LIN {X 0,Y 544.562,Z 1211.677,A -85,B 0,C 180,E1 25546.246,E2 25546.246} C_VEL
LIN {X 0,Y 545.068,Z 1204.229,A -85,B 0,C 180,E1 25544.028,E2 25544.028} C_VEL
LIN {X 0,Y 545.864,Z 1194.826,A -85,B 0,C 180,E1 25541.746,E2 25541.746} C_VEL
LIN {X 0,Y 546.932,Z 1184.101,A -85,B 0,C 180,E1 25539.563,E2 25539.563} C_VEL
LIN {X 0,Y 548.229,Z 1171.822,A -85,B 0,C 180,E1 25537.48,E2 25537.48} C_VEL
LIN {X 0,Y 549.884,Z 1157.402,A -85,B 0,C 180,E1 25535.392,E2 25535.392} C_VEL
LIN {X 0,Y 551.64,Z 1142.682,A -85,B 0,C 180,E1 25533.563,E2 25533.563} C_VEL
LIN {X 0,Y 553.416,Z 1127.177,A -85,B 0,C 180,E1 25531.923,E2 25531.923} C_VEL
LIN {X 0,Y 555.29,Z 1110.35,A -85,B 0,C 180,E1 25530.377,E2 25530.377} C_VEL
LIN {X 0,Y 557.037,Z 1093.4,A -85,B 0,C 180,E1 25529.051,E2 25529.051} C_VEL
LIN {X 0,Y 558.861,Z 1073.803,A -85,B 0,C 180,E1 25527.747,E2 25527.747} C_VEL
LIN {X 0,Y 560.413,Z 1054.46,A -85,B 0,C 180,E1 25526.665,E2 25526.665} C_VEL
LIN {X 0,Y 561.698,Z 1033.944,A -85,B 0,C 180,E1 25525.739,E2 25525.739} C_VEL
LIN {X 0,Y 562.756,Z 1011.905,A -85,B 0,C 180,E1 25524.95,E2 25524.95} C_VEL
LIN {X 0,Y 563.403,Z 990.948,A -85,B 0,C 180,E1 25524.379,E2 25524.379} C_VEL
LIN {X 0,Y 563.645,Z 969.284,A -85,B 0,C 180,E1 25523.981,E2 25523.981} C_VEL
LIN {X 0,Y 565.376,Z 853.6,A -85,B 0,C 180,E1 25522.448,E2 25522.448} C_VEL
LIN {X 0,Y 567.818,Z 763.974,A -85,B 0,C 180,E1 25521.099,E2 25521.099} C_VEL
LIN {X 0,Y 569.634,Z 711.383,A -85,B 0,C 180,E1 25520.211,E2 25520.211} C_VEL
LIN {X 0,Y 564.325,Z 714.5,A -85,B 0,C 180,E1 25519.789,E2 25519.789} C_VEL
LIN {X 0,Y 560.672,Z 715.375,A -85,B 0,C 180,E1 25519.441,E2 25519.441} C_VEL
LIN {X 0,Y 559.123,Z 715.198,A -85,B 0,C 180,E1 25519.252,E2 25519.252} C_VEL
LIN {X 0,Y 554.906,Z 729.11,A -85,B 0,C 180,E1 25517.706,E2 25517.706} C_VEL
LIN {X 0,Y 551.52,Z 746.313,A -85,B 0,C 180,E1 25516.035,E2 25516.035} C_VEL
LIN {X 0,Y 548.829,Z 768.841,A -85,B 0,C 180,E1 25514.104,E2 25514.104} C_VEL
LIN {X 0,Y 548.008,Z 793.1,A -85,B 0,C 180,E1 25512.18,E2 25512.18} C_VEL
LIN {X 0,Y 549.552,Z 814.095,A -85,B 0,C 180,E1 25510.568,E2 25510.568} C_VEL
LIN {X 0,Y 553.126,Z 833.312,A -85,B 0,C 180,E1 25509.117,E2 25509.117} C_VEL
LIN {X 0,Y 558.641,Z 851.04,A -85,B 0,C 180,E1 25507.793,E2 25507.793} C_VEL
LIN {X 0,Y 566.486,Z 868.661,A -85,B 0,C 180,E1 25506.502,E2 25506.502} C_VEL
LIN {X 0,Y 575.748,Z 884.402,A -85,B 0,C 180,E1 25505.375,E2 25505.375} C_VEL
LIN {X 0,Y 586.391,Z 898.731,A -85,B 0,C 180,E1 25504.381,E2 25504.381} C_VEL
LIN {X 0,Y 587.254,Z 899.863,A -85,B 0,C 180,E1 25504.305,E2 25504.305} C_VEL
LIN {X 0,Y 579.576,Z 911.271,A -85,B 0,C 180,E1 25503.697,E2 25503.697} C_VEL
LIN {X 0,Y 571.301,Z 934.87,A -85,B 0,C 180,E1 25503.762,E2 25503.762} C_VEL
LIN {X 0,Y 566.013,Z 954.731,A -85,B 0,C 180,E1 25503.715,E2 25503.715} C_VEL
LIN {X 0,Y 563.46,Z 969.81,A -85,B 0,C 180,E1 25503.539,E2 25503.539} C_VEL
LIN {X 0,Y 562.158,Z 989.948,A -85,B 0,C 180,E1 25503.128,E2 25503.128} C_VEL
LIN {X 0,Y 560.251,Z 1022.157,A -85,B 0,C 180,E1 25502.29,E2 25502.29} C_VEL
LIN {X 0,Y 558.395,Z 1051.426,A -85,B 0,C 180,E1 25501.335,E2 25501.335} C_VEL
LIN {X 0,Y 556.632,Z 1080.044,A -85,B 0,C 180,E1 25500.198,E2 25500.198} C_VEL
LIN {X 0,Y 554.956,Z 1107.84,A -85,B 0,C 180,E1 25498.874,E2 25498.874} C_VEL
LIN {X 0,Y 553.378,Z 1132.67,A -85,B 0,C 180,E1 25497.478,E2 25497.478} C_VEL
LIN {X 0,Y 551.863,Z 1155.997,A -85,B 0,C 180,E1 25495.948,E2 25495.948} C_VEL
LIN {X 0,Y 550.467,Z 1176.831,A -85,B 0,C 180,E1 25494.353,E2 25494.353} C_VEL
LIN {X 0,Y 549.066,Z 1196.682,A -85,B 0,C 180,E1 25492.588,E2 25492.588} C_VEL
LIN {X 0,Y 547.917,Z 1213.443,A -85,B 0,C 180,E1 25490.847,E2 25490.847} C_VEL
LIN {X 0,Y 546.809,Z 1229.626,A -85,B 0,C 180,E1 25488.886,E2 25488.886} C_VEL
LIN {X 0,Y 545.96,Z 1242.613,A -85,B 0,C 180,E1 25487.041,E2 25487.041} C_VEL
LIN {X 0,Y 545.256,Z 1254.791,A -85,B 0,C 180,E1 25484.986,E2 25484.986} C_VEL
LIN {X 0,Y 544.689,Z 1265.458,A -85,B 0,C 180,E1 25482.835,E2 25482.835} C_VEL
LIN {X 0,Y 544.341,Z 1274.037,A -85,B 0,C 180,E1 25480.693,E2 25480.693} C_VEL
LIN {X 0,Y 544.118,Z 1281.473,A -85,B 0,C 180,E1 25478.349,E2 25478.349} C_VEL
LIN {X 0,Y 544.015,Z 1286.703,A -85,B 0,C 180,E1 25476.092,E2 25476.092} C_VEL
LIN {X 0,Y 543.973,Z 1290.229,A -85,B 0,C 180,E1 25473.901,E2 25473.901} C_VEL
LIN {X 0,Y 543.96,Z 1292.291,A -85,B 0,C 180,E1 25471.581,E2 25471.581} C_VEL
LIN {X 0,Y 543.956,Z 1292.686,A -85,B 0,C 180,E1 25469.264,E2 25469.264} C_VEL
LIN {X 0,Y 543.956,Z 1291.533,A -85,B 0,C 180,E1 25467.051,E2 25467.051} C_VEL
LIN {X 0,Y 543.973,Z 1288.582,A -85,B 0,C 180,E1 25464.622,E2 25464.622} C_VEL
LIN {X 0,Y 544.03,Z 1284.043,A -85,B 0,C 180,E1 25462.291,E2 25462.291} C_VEL
LIN {X 0,Y 544.211,Z 1277.901,A -85,B 0,C 180,E1 25460,E2 25460} C_VEL
LIN {X 0,Y 544.557,Z 1270.094,A -85,B 0,C 180,E1 25457.704,E2 25457.704} C_VEL
LIN {X 0,Y 545.171,Z 1259.584,A -85,B 0,C 180,E1 25455.232,E2 25455.232} C_VEL
LIN {X 0,Y 546.016,Z 1247.891,A -85,B 0,C 180,E1 25452.964,E2 25452.964} C_VEL
LIN {X 0,Y 547.133,Z 1234.759,A -85,B 0,C 180,E1 25450.797,E2 25450.797} C_VEL
LIN {X 0,Y 548.623,Z 1219.348,A -85,B 0,C 180,E1 25448.624,E2 25448.624} C_VEL
LIN {X 0,Y 550.417,Z 1202.151,A -85,B 0,C 180,E1 25446.547,E2 25446.547} C_VEL
LIN {X 0,Y 552.431,Z 1184.117,A -85,B 0,C 180,E1 25444.664,E2 25444.664} C_VEL
LIN {X 0,Y 554.712,Z 1164.306,A -85,B 0,C 180,E1 25442.87,E2 25442.87} C_VEL
LIN {X 0,Y 556.979,Z 1144.891,A -85,B 0,C 180,E1 25441.361,E2 25441.361} C_VEL
LIN {X 0,Y 559.484,Z 1123.679,A -85,B 0,C 180,E1 25439.916,E2 25439.916} C_VEL
LIN {X 0,Y 562.031,Z 1101.534,A -85,B 0,C 180,E1 25438.645,E2 25438.645} C_VEL
LIN {X 0,Y 564.568,Z 1079.231,A -85,B 0,C 180,E1 25437.547,E2 25437.547} C_VEL
LIN {X 0,Y 567.05,Z 1055.53,A -85,B 0,C 180,E1 25436.599,E2 25436.599} C_VEL
LIN {X 0,Y 569.474,Z 1031.429,A -85,B 0,C 180,E1 25435.818,E2 25435.818} C_VEL
LIN {X 0,Y 571.497,Z 1007.453,A -85,B 0,C 180,E1 25435.234,E2 25435.234} C_VEL
LIN {X 0,Y 573.01,Z 980.269,A -85,B 0,C 180,E1 25434.735,E2 25434.735} C_VEL
LIN {X 0,Y 574.653,Z 963.231,A -85,B 0,C 180,E1 25434.528,E2 25434.528} C_VEL
LIN {X 0,Y 576.296,Z 952.9,A -85,B 0,C 180,E1 25434.434,E2 25434.434} C_VEL
LIN {X 0,Y 584.411,Z 939.055,A -85,B 0,C 180,E1 25433.704,E2 25433.704} C_VEL
LIN {X 0,Y 595.54,Z 921.987,A -85,B 0,C 180,E1 25432.893,E2 25432.893} C_VEL
LIN {X 0,Y 595.784,Z 921.452,A -85,B 0,C 180,E1 25432.862,E2 25432.862} C_VEL
LIN {X 0,Y 586.983,Z 910.439,A -85,B 0,C 180,E1 25431.433,E2 25431.433} C_VEL
LIN {X 0,Y 579.494,Z 897.396,A -85,B 0,C 180,E1 25429.852,E2 25429.852} C_VEL
LIN {X 0,Y 573.88,Z 882.911,A -85,B 0,C 180,E1 25428.221,E2 25428.221} C_VEL
LIN {X 0,Y 570.376,Z 867.493,A -85,B 0,C 180,E1 25426.595,E2 25426.595} C_VEL
LIN {X 0,Y 568.831,Z 850.15,A -85,B 0,C 180,E1 25424.898,E2 25424.898} C_VEL
LIN {X 0,Y 569.395,Z 830.215,A -85,B 0,C 180,E1 25423.073,E2 25423.073} C_VEL
LIN {X 0,Y 573.141,Z 791.098,A -85,B 0,C 180,E1 25419.636,E2 25419.636} C_VEL
LIN {X 0,Y 576.634,Z 756.144,A -85,B 0,C 180,E1 25416.496,E2 25416.496} C_VEL
LIN {X 0,Y 579.993,Z 723.11,A -85,B 0,C 180,E1 25413.45,E2 25413.45} C_VEL
LIN {X 0,Y 581.981,Z 702.852,A -85,B 0,C 180,E1 25411.527,E2 25411.527} C_VEL
LIN {X 0,Y 573.862,Z 683.052,A -85,B 0,C 180,E1 25408.517,E2 25408.517} C_VEL
LIN {X 0,Y 566.014,Z 664.757,A -85,B 0,C 180,E1 25405.534,E2 25405.534} C_VEL
LIN {X 0,Y 558.284,Z 647.753,A -85,B 0,C 180,E1 25402.537,E2 25402.537} C_VEL
LIN {X 0,Y 552.535,Z 635.448,A -85,B 0,C 180,E1 25400.221,E2 25400.221} C_VEL
LIN {X 0,Y 549.142,Z 628.134,A -85,B 0,C 180,E1 25398.801,E2 25398.801} C_VEL
LIN {X 0,Y 547.28,Z 624.068,A -85,B 0,C 180,E1 25397.985,E2 25397.985} C_VEL
LIN {X 0,Y 545.723,Z 620.923,A -85,B 0,C 180,E1 25397.34,E2 25397.34} C_VEL
LIN {X 0,Y 545.56,Z 620.018,A -85,B 0,C 180,E1 25397.162,E2 25397.162} C_VEL
LIN {X 0,Y 545.561,Z 620.023,A -85,B 0,C 180,E1 25393.676,E2 25393.676} C_VEL
LIN {X 0,Y 545.551,Z 620.018,A -85,B 0,C 180,E1 25390.347,E2 25390.347} C_VEL
LIN {X 0,Y 545.565,Z 620.021,A -85,B 0,C 180,E1 25386.948,E2 25386.948} C_VEL
LIN {X 0,Y 545.556,Z 620.018,A -85,B 0,C 180,E1 25383.573,E2 25383.573} C_VEL
LIN {X 0,Y 545.556,Z 620.024,A -85,B 0,C 180,E1 25380.21,E2 25380.21} C_VEL
LIN {X 0,Y 545.55,Z 620.025,A -85,B 0,C 180,E1 25376.848,E2 25376.848} C_VEL
LIN {X 0,Y 545.559,Z 620.021,A -85,B 0,C 180,E1 25373.475,E2 25373.475} C_VEL
LIN {X 0,Y 545.558,Z 620.018,A -85,B 0,C 180,E1 25369.973,E2 25369.973} C_VEL
LIN {X 0,Y 545.56,Z 620.016,A -85,B 0,C 180,E1 25366.54,E2 25366.54} C_VEL
LIN {X 0,Y 545.551,Z 620.018,A -85,B 0,C 180,E1 25363.277,E2 25363.277} C_VEL
LIN {X 0,Y 545.563,Z 620.017,A -85,B 0,C 180,E1 25359.957,E2 25359.957} C_VEL
LIN {X 0,Y 545.562,Z 620.016,A -85,B 0,C 180,E1 25356.565,E2 25356.565} C_VEL
LIN {X 0,Y 545.555,Z 620.015,A -85,B 0,C 180,E1 25353.193,E2 25353.193} C_VEL
LIN {X 0,Y 545.551,Z 620.019,A -85,B 0,C 180,E1 25349.855,E2 25349.855} C_VEL
LIN {X 0,Y 545.558,Z 620.022,A -85,B 0,C 180,E1 25346.499,E2 25346.499} C_VEL
LIN {X 0,Y 545.561,Z 620.023,A -85,B 0,C 180,E1 25343.04,E2 25343.04} C_VEL
LIN {X 0,Y 545.564,Z 620.024,A -85,B 0,C 180,E1 25339.676,E2 25339.676} C_VEL
LIN {X 0,Y 545.549,Z 619.992,A -85,B 0,C 180,E1 25336.293,E2 25336.293} C_VEL
LIN {X 0,Y 545.561,Z 620.016,A -85,B 0,C 180,E1 25332.981,E2 25332.981} C_VEL
LIN {X 0,Y 545.567,Z 620.029,A -85,B 0,C 180,E1 25329.625,E2 25329.625} C_VEL
LIN {X 0,Y 545.579,Z 620.17,A -85,B 0,C 180,E1 25326.359,E2 25326.359} C_VEL
LIN {X 0,Y 554.088,Z 644.386,A -85,B 0,C 180,E1 25324.075,E2 25324.075} C_VEL
LIN {X 0,Y 559.543,Z 662.583,A -85,B 0,C 180,E1 25322.416,E2 25322.416} C_VEL
LIN {X 0,Y 558.089,Z 702.519,A -85,B 0,C 180,E1 25319.516,E2 25319.516} C_VEL
LIN {X 0,Y 556.154,Z 749.591,A -85,B 0,C 180,E1 25316.075,E2 25316.075} C_VEL
LIN {X 0,Y 554.34,Z 796.346,A -85,B 0,C 180,E1 25312.704,E2 25312.704} C_VEL
LIN {X 0,Y 553.05,Z 840.958,A -85,B 0,C 180,E1 25309.618,E2 25309.618} C_VEL
LIN {X 0,Y 553.037,Z 845.924,A -85,B 0,C 180,E1 25309.313,E2 25309.313} C_VEL
LIN {X 0,Y 553.774,Z 853.842,A -85,B 0,C 180,E1 25309.176,E2 25309.176} C_VEL
LIN {X 0,Y 553.745,Z 856.037,A -85,B 0,C 180,E1 25309.148,E2 25309.148} C_VEL
LIN {X 0,Y 552.713,Z 863.711,A -85,B 0,C 180,E1 25309.083,E2 25309.083} C_VEL
LIN {X 0,Y 546.531,Z 884.049,A -85,B 0,C 180,E1 25309.045,E2 25309.045} C_VEL
LIN {X 0,Y 545.779,Z 890.637,A -85,B 0,C 180,E1 25308.984,E2 25308.984} C_VEL
LIN {X 0,Y 544.332,Z 1016.575,A -85,B 0,C 180,E1 25307.282,E2 25307.282} C_VEL
LIN {X 0,Y 544.07,Z 1034.06,A -85,B 0,C 180,E1 25306.854,E2 25306.854} C_VEL
LIN {X 0,Y 543.55,Z 1050.898,A -85,B 0,C 180,E1 25306.235,E2 25306.235} C_VEL
LIN {X 0,Y 542.849,Z 1067.086,A -85,B 0,C 180,E1 25305.434,E2 25305.434} C_VEL
LIN {X 0,Y 542.02,Z 1082.23,A -85,B 0,C 180,E1 25304.474,E2 25304.474} C_VEL
LIN {X 0,Y 541.114,Z 1096.279,A -85,B 0,C 180,E1 25303.353,E2 25303.353} C_VEL
LIN {X 0,Y 540.183,Z 1109.272,A -85,B 0,C 180,E1 25302.072,E2 25302.072} C_VEL
LIN {X 0,Y 539.316,Z 1120.771,A -85,B 0,C 180,E1 25300.683,E2 25300.683} C_VEL
LIN {X 0,Y 538.552,Z 1130.856,A -85,B 0,C 180,E1 25299.186,E2 25299.186} C_VEL
LIN {X 0,Y 537.911,Z 1139.49,A -85,B 0,C 180,E1 25297.582,E2 25297.582} C_VEL
LIN {X 0,Y 537.417,Z 1146.684,A -85,B 0,C 180,E1 25295.872,E2 25295.872} C_VEL
LIN {X 0,Y 537.07,Z 1152.376,A -85,B 0,C 180,E1 25294.055,E2 25294.055} C_VEL
LIN {X 0,Y 536.865,Z 1156.258,A -85,B 0,C 180,E1 25292.24,E2 25292.24} C_VEL
LIN {X 0,Y 536.762,Z 1158.468,A -85,B 0,C 180,E1 25290.319,E2 25290.319} C_VEL
LIN {X 0,Y 536.741,Z 1158.887,A -85,B 0,C 180,E1 25288.397,E2 25288.397} C_VEL
LIN {X 0,Y 536.82,Z 1157.529,A -85,B 0,C 180,E1 25286.475,E2 25286.475} C_VEL
LIN {X 0,Y 536.987,Z 1154.493,A -85,B 0,C 180,E1 25284.657,E2 25284.657} C_VEL
LIN {X 0,Y 537.286,Z 1149.689,A -85,B 0,C 180,E1 25282.836,E2 25282.836} C_VEL
LIN {X 0,Y 537.745,Z 1142.99,A -85,B 0,C 180,E1 25281.013,E2 25281.013} C_VEL
LIN {X 0,Y 538.329,Z 1135.257,A -85,B 0,C 180,E1 25279.403,E2 25279.403} C_VEL
LIN {X 0,Y 539.094,Z 1125.43,A -85,B 0,C 180,E1 25277.792,E2 25277.792} C_VEL
LIN {X 0,Y 539.999,Z 1114.033,A -85,B 0,C 180,E1 25276.289,E2 25276.289} C_VEL
LIN {X 0,Y 540.962,Z 1101.428,A -85,B 0,C 180,E1 25274.939,E2 25274.939} C_VEL
LIN {X 0,Y 541.899,Z 1087.841,A -85,B 0,C 180,E1 25273.766,E2 25273.766} C_VEL
LIN {X 0,Y 542.778,Z 1073.195,A -85,B 0,C 180,E1 25272.746,E2 25272.746} C_VEL
LIN {X 0,Y 543.555,Z 1057.58,A -85,B 0,C 180,E1 25271.886,E2 25271.886} C_VEL
LIN {X 0,Y 544.156,Z 1041.565,A -85,B 0,C 180,E1 25271.213,E2 25271.213} C_VEL
LIN {X 0,Y 544.545,Z 1024.25,A -85,B 0,C 180,E1 25270.701,E2 25270.701} C_VEL
LIN {X 0,Y 544.693,Z 1004.749,A -85,B 0,C 180,E1 25270.351,E2 25270.351} C_VEL
LIN {X 0,Y 546.455,Z 851.134,A -85,B 0,C 180,E1 25268.298,E2 25268.298} C_VEL
LIN {X 0,Y 545.809,Z 845.842,A -85,B 0,C 180,E1 25268.167,E2 25268.167} C_VEL
LIN {X 0,Y 547.153,Z 801.476,A -85,B 0,C 180,E1 25265.087,E2 25265.087} C_VEL
LIN {X 0,Y 548.938,Z 757.8,A -85,B 0,C 180,E1 25261.909,E2 25261.909} C_VEL
LIN {X 0,Y 550.971,Z 712.063,A -85,B 0,C 180,E1 25258.534,E2 25258.534} C_VEL
LIN {X 0,Y 552.718,Z 669.961,A -85,B 0,C 180,E1 25255.442,E2 25255.442} C_VEL
LIN {X 0,Y 552.763,Z 665.3,A -85,B 0,C 180,E1 25255.094,E2 25255.094} C_VEL
LIN {X 0,Y 545.767,Z 643.324,A -85,B 0,C 180,E1 25253.015,E2 25253.015} C_VEL
LIN {X 0,Y 538.244,Z 623.221,A -85,B 0,C 180,E1 25251.028,E2 25251.028} C_VEL
LIN {X 0,Y 537.625,Z 620.99,A -85,B 0,C 180,E1 25250.81,E2 25250.81} C_VEL
LIN {X 0,Y 537.624,Z 621.01,A -85,B 0,C 180,E1 25247.391,E2 25247.391} C_VEL
LIN {X 0,Y 537.619,Z 621.012,A -85,B 0,C 180,E1 25243.926,E2 25243.926} C_VEL
LIN {X 0,Y 537.636,Z 621.101,A -85,B 0,C 180,E1 25241.577,E2 25241.577} C_VEL
LIN {X 0,Y 539.132,Z 624.777,A -85,B 0,C 180,E1 25240.988,E2 25240.988} C_VEL
LIN {X 0,Y 544.561,Z 636.539,A -85,B 0,C 180,E1 25239.145,E2 25239.145} C_VEL
LIN {X 0,Y 562.473,Z 662.364,A -85,B 0,C 180,E1 25237.043,E2 25237.043} C_VEL
LIN {X 0,Y 572.59,Z 677.716,A -85,B 0,C 180,E1 25235.923,E2 25235.923} C_VEL
LIN {X 0,Y 563.214,Z 919.475,A -85,B 0,C 180,E1 25232.101,E2 25232.101} C_VEL
LIN {X 0,Y 561.649,Z 966.293,A -85,B 0,C 180,E1 25231.336,E2 25231.336} C_VEL
LIN {X 0,Y 560.501,Z 989.145,A -85,B 0,C 180,E1 25230.77,E2 25230.77} C_VEL
LIN {X 0,Y 559.003,Z 1011.643,A -85,B 0,C 180,E1 25230.032,E2 25230.032} C_VEL
LIN {X 0,Y 557.268,Z 1033.005,A -85,B 0,C 180,E1 25229.153,E2 25229.153} C_VEL
LIN {X 0,Y 555.198,Z 1053.829,A -85,B 0,C 180,E1 25228.096,E2 25228.096} C_VEL
LIN {X 0,Y 552.898,Z 1075.118,A -85,B 0,C 180,E1 25226.804,E2 25226.804} C_VEL
LIN {X 0,Y 550.629,Z 1094.218,A -85,B 0,C 180,E1 25225.434,E2 25225.434} C_VEL
LIN {X 0,Y 548.259,Z 1112.608,A -85,B 0,C 180,E1 25223.883,E2 25223.883} C_VEL
LIN {X 0,Y 545.977,Z 1130.204,A -85,B 0,C 180,E1 25222.164,E2 25222.164} C_VEL
LIN {X 0,Y 543.939,Z 1145.349,A -85,B 0,C 180,E1 25220.443,E2 25220.443} C_VEL
LIN {X 0,Y 541.915,Z 1160.932,A -85,B 0,C 180,E1 25218.392,E2 25218.392} C_VEL
LIN {X 0,Y 540.25,Z 1174.381,A -85,B 0,C 180,E1 25216.339,E2 25216.339} C_VEL
LIN {X 0,Y 538.865,Z 1186.313,A -85,B 0,C 180,E1 25214.178,E2 25214.178} C_VEL
LIN {X 0,Y 537.78,Z 1196.995,A -85,B 0,C 180,E1 25211.91,E2 25211.91} C_VEL
LIN {X 0,Y 537.051,Z 1205.44,A -85,B 0,C 180,E1 25209.754,E2 25209.754} C_VEL
LIN {X 0,Y 536.512,Z 1213.345,A -85,B 0,C 180,E1 25207.281,E2 25207.281} C_VEL
LIN {X 0,Y 536.226,Z 1218.992,A -85,B 0,C 180,E1 25205.028,E2 25205.028} C_VEL
LIN {X 0,Y 536.064,Z 1223.49,A -85,B 0,C 180,E1 25202.566,E2 25202.566} C_VEL
LIN {X 0,Y 536.028,Z 1226.336,A -85,B 0,C 180,E1 25200.214,E2 25200.214} C_VEL
LIN {X 0,Y 535.991,Z 1227.612,A -85,B 0,C 180,E1 25197.862,E2 25197.862} C_VEL
LIN {X 0,Y 535.993,Z 1227.555,A -85,B 0,C 180,E1 25195.506,E2 25195.506} C_VEL
LIN {X 0,Y 536.023,Z 1225.893,A -85,B 0,C 180,E1 25193.143,E2 25193.143} C_VEL
LIN {X 0,Y 536.112,Z 1222.854,A -85,B 0,C 180,E1 25190.77,E2 25190.77} C_VEL
LIN {X 0,Y 536.279,Z 1218.382,A -85,B 0,C 180,E1 25188.492,E2 25188.492} C_VEL
LIN {X 0,Y 536.653,Z 1211.807,A -85,B 0,C 180,E1 25185.983,E2 25185.983} C_VEL
LIN {X 0,Y 537.235,Z 1204.125,A -85,B 0,C 180,E1 25183.678,E2 25183.678} C_VEL
LIN {X 0,Y 538.089,Z 1194.661,A -85,B 0,C 180,E1 25181.389,E2 25181.389} C_VEL
LIN {X 0,Y 539.201,Z 1184.229,A -85,B 0,C 180,E1 25179.256,E2 25179.256} C_VEL
LIN {X 0,Y 540.599,Z 1171.911,A -85,B 0,C 180,E1 25177.144,E2 25177.144} C_VEL
LIN {X 0,Y 542.265,Z 1158.093,A -85,B 0,C 180,E1 25175.124,E2 25175.124} C_VEL
LIN {X 0,Y 544.124,Z 1143.344,A -85,B 0,C 180,E1 25173.264,E2 25173.264} C_VEL
LIN {X 0,Y 546.025,Z 1127.486,A -85,B 0,C 180,E1 25171.568,E2 25171.568} C_VEL
LIN {X 0,Y 548.147,Z 1109.199,A -85,B 0,C 180,E1 25169.892,E2 25169.892} C_VEL
LIN {X 0,Y 550.104,Z 1091.165,A -85,B 0,C 180,E1 25168.483,E2 25168.483} C_VEL
LIN {X 0,Y 551.853,Z 1072.399,A -85,B 0,C 180,E1 25167.259,E2 25167.259} C_VEL
LIN {X 0,Y 553.498,Z 1051.713,A -85,B 0,C 180,E1 25166.13,E2 25166.13} C_VEL
LIN {X 0,Y 554.841,Z 1031.303,A -85,B 0,C 180,E1 25165.224,E2 25165.224} C_VEL
LIN {X 0,Y 555.771,Z 1010.369,A -85,B 0,C 180,E1 25164.503,E2 25164.503} C_VEL
LIN {X 0,Y 556.37,Z 988.036,A -85,B 0,C 180,E1 25163.928,E2 25163.928} C_VEL
LIN {X 0,Y 556.586,Z 965.593,A -85,B 0,C 180,E1 25163.54,E2 25163.54} C_VEL
LIN {X 0,Y 558.266,Z 867.649,A -85,B 0,C 180,E1 25162.215,E2 25162.215} C_VEL
LIN {X 0,Y 560.827,Z 781.835,A -85,B 0,C 180,E1 25160.892,E2 25160.892} C_VEL
LIN {X 0,Y 563.225,Z 722.74,A -85,B 0,C 180,E1 25159.87,E2 25159.87} C_VEL
LIN {X 0,Y 559.432,Z 723.517,A -85,B 0,C 180,E1 25159.51,E2 25159.51} C_VEL
LIN {X 0,Y 553.862,Z 727.441,A -85,B 0,C 180,E1 25158.993,E2 25158.993} C_VEL
LIN {X 0,Y 550.494,Z 728.74,A -85,B 0,C 180,E1 25158.605,E2 25158.605} C_VEL
LIN {X 0,Y 549.002,Z 728.818,A -85,B 0,C 180,E1 25158.387,E2 25158.387} C_VEL
LIN {X 0,Y 545.176,Z 744.683,A -85,B 0,C 180,E1 25156.731,E2 25156.731} C_VEL
LIN {X 0,Y 542.101,Z 764.837,A -85,B 0,C 180,E1 25154.879,E2 25154.879} C_VEL
LIN {X 0,Y 540.482,Z 788.554,A -85,B 0,C 180,E1 25152.895,E2 25152.895} C_VEL
LIN {X 0,Y 541.18,Z 809.258,A -85,B 0,C 180,E1 25151.238,E2 25151.238} C_VEL
LIN {X 0,Y 543.953,Z 828.754,A -85,B 0,C 180,E1 25149.71,E2 25149.71} C_VEL
LIN {X 0,Y 548.863,Z 847.38,A -85,B 0,C 180,E1 25148.273,E2 25148.273} C_VEL
LIN {X 0,Y 555.897,Z 865.129,A -85,B 0,C 180,E1 25146.926,E2 25146.926} C_VEL
LIN {X 0,Y 564.621,Z 881.535,A -85,B 0,C 180,E1 25145.712,E2 25145.712} C_VEL
LIN {X 0,Y 574.804,Z 896.536,A -85,B 0,C 180,E1 25144.634,E2 25144.634} C_VEL
LIN {X 0,Y 577.615,Z 900.54,A -85,B 0,C 180,E1 25144.357,E2 25144.357} C_VEL
LIN {X 0,Y 574.007,Z 906.053,A -85,B 0,C 180,E1 25144.075,E2 25144.075} C_VEL
LIN {X 0,Y 564.767,Z 932.57,A -85,B 0,C 180,E1 25144.167,E2 25144.167} C_VEL
LIN {X 0,Y 559.323,Z 952.643,A -85,B 0,C 180,E1 25144.117,E2 25144.117} C_VEL
LIN {X 0,Y 556.547,Z 967.971,A -85,B 0,C 180,E1 25143.939,E2 25143.939} C_VEL
LIN {X 0,Y 555.208,Z 984.466,A -85,B 0,C 180,E1 25143.603,E2 25143.603} C_VEL
LIN {X 0,Y 553.15,Z 1017.086,A -85,B 0,C 180,E1 25142.748,E2 25142.748} C_VEL
LIN {X 0,Y 551.133,Z 1046.801,A -85,B 0,C 180,E1 25141.776,E2 25141.776} C_VEL
LIN {X 0,Y 549.282,Z 1075.281,A -85,B 0,C 180,E1 25140.645,E2 25140.645} C_VEL
LIN {X 0,Y 547.548,Z 1102.102,A -85,B 0,C 180,E1 25139.379,E2 25139.379} C_VEL
LIN {X 0,Y 545.849,Z 1128.091,A -85,B 0,C 180,E1 25137.934,E2 25137.934} C_VEL
LIN {X 0,Y 544.224,Z 1152.54,A -85,B 0,C 180,E1 25136.341,E2 25136.341} C_VEL
LIN {X 0,Y 542.747,Z 1173.837,A -85,B 0,C 180,E1 25134.722,E2 25134.722} C_VEL
LIN {X 0,Y 541.3,Z 1194,A -85,B 0,C 180,E1 25132.941,E2 25132.941} C_VEL
LIN {X 0,Y 540.13,Z 1210.759,A -85,B 0,C 180,E1 25131.219,E2 25131.219} C_VEL
LIN {X 0,Y 539.005,Z 1226.92,A -85,B 0,C 180,E1 25129.282,E2 25129.282} C_VEL
LIN {X 0,Y 538.056,Z 1241.043,A -85,B 0,C 180,E1 25127.299,E2 25127.299} C_VEL
LIN {X 0,Y 537.314,Z 1253.479,A -85,B 0,C 180,E1 25125.213,E2 25125.213} C_VEL
LIN {X 0,Y 536.73,Z 1264.436,A -85,B 0,C 180,E1 25123.013,E2 25123.013} C_VEL
LIN {X 0,Y 536.367,Z 1273.129,A -85,B 0,C 180,E1 25120.854,E2 25120.854} C_VEL
LIN {X 0,Y 536.145,Z 1280.396,A -85,B 0,C 180,E1 25118.582,E2 25118.582} C_VEL
LIN {X 0,Y 536.036,Z 1285.812,A -85,B 0,C 180,E1 25116.32,E2 25116.32} C_VEL
LIN {X 0,Y 535.988,Z 1289.677,A -85,B 0,C 180,E1 25113.959,E2 25113.959} C_VEL
LIN {X 0,Y 535.978,Z 1291.733,A -85,B 0,C 180,E1 25111.712,E2 25111.712} C_VEL
LIN {X 0,Y 535.97,Z 1292.217,A -85,B 0,C 180,E1 25109.253,E2 25109.253} C_VEL
LIN {X 0,Y 535.968,Z 1291.077,A -85,B 0,C 180,E1 25107.007,E2 25107.007} C_VEL
LIN {X 0,Y 535.979,Z 1288.087,A -85,B 0,C 180,E1 25104.542,E2 25104.542} C_VEL
LIN {X 0,Y 536.036,Z 1283.513,A -85,B 0,C 180,E1 25102.175,E2 25102.175} C_VEL
LIN {X 0,Y 536.234,Z 1277.177,A -85,B 0,C 180,E1 25099.798,E2 25099.798} C_VEL
LIN {X 0,Y 536.587,Z 1269.432,A -85,B 0,C 180,E1 25097.518,E2 25097.518} C_VEL
LIN {X 0,Y 537.237,Z 1258.85,A -85,B 0,C 180,E1 25095.006,E2 25095.006} C_VEL
LIN {X 0,Y 538.181,Z 1246.475,A -85,B 0,C 180,E1 25092.597,E2 25092.597} C_VEL
LIN {X 0,Y 539.379,Z 1233.108,A -85,B 0,C 180,E1 25090.397,E2 25090.397} C_VEL
LIN {X 0,Y 540.965,Z 1217.481,A -85,B 0,C 180,E1 25088.193,E2 25088.193} C_VEL
LIN {X 0,Y 543.005,Z 1199.051,A -85,B 0,C 180,E1 25085.971,E2 25085.971} C_VEL
LIN {X 0,Y 545.361,Z 1178.845,A -85,B 0,C 180,E1 25083.896,E2 25083.896} C_VEL
LIN {X 0,Y 547.773,Z 1158.882,A -85,B 0,C 180,E1 25082.143,E2 25082.143} C_VEL
LIN {X 0,Y 550.131,Z 1139.735,A -85,B 0,C 180,E1 25080.673,E2 25080.673} C_VEL
LIN {X 0,Y 552.94,Z 1116.823,A -85,B 0,C 180,E1 25079.161,E2 25079.161} C_VEL
LIN {X 0,Y 555.352,Z 1097.015,A -85,B 0,C 180,E1 25078.042,E2 25078.042} C_VEL
LIN {X 0,Y 558.237,Z 1071.944,A -85,B 0,C 180,E1 25076.851,E2 25076.851} C_VEL
LIN {X 0,Y 560.724,Z 1049.643,A -85,B 0,C 180,E1 25075.985,E2 25075.985} C_VEL
LIN {X 0,Y 563.233,Z 1024.721,A -85,B 0,C 180,E1 25075.219,E2 25075.219} C_VEL
LIN {X 0,Y 565.241,Z 1001.127,A -85,B 0,C 180,E1 25074.661,E2 25074.661} C_VEL
LIN {X 0,Y 566.987,Z 972.381,A -85,B 0,C 180,E1 25074.169,E2 25074.169} C_VEL
LIN {X 0,Y 569.907,Z 951.51,A -85,B 0,C 180,E1 25073.971,E2 25073.971} C_VEL
LIN {X 0,Y 578.073,Z 937.676,A -85,B 0,C 180,E1 25073.242,E2 25073.242} C_VEL
LIN {X 0,Y 586.981,Z 923.541,A -85,B 0,C 180,E1 25072.543,E2 25072.543} C_VEL
LIN {X 0,Y 578.464,Z 912.034,A -85,B 0,C 180,E1 25071.063,E2 25071.063} C_VEL
LIN {X 0,Y 571.261,Z 898.435,A -85,B 0,C 180,E1 25069.433,E2 25069.433} C_VEL
LIN {X 0,Y 566.009,Z 883.482,A -85,B 0,C 180,E1 25067.748,E2 25067.748} C_VEL
LIN {X 0,Y 562.857,Z 867.576,A -85,B 0,C 180,E1 25066.084,E2 25066.084} C_VEL
LIN {X 0,Y 561.725,Z 849.486,A -85,B 0,C 180,E1 25064.313,E2 25064.313} C_VEL
LIN {X 0,Y 562.737,Z 828.652,A -85,B 0,C 180,E1 25062.418,E2 25062.418} C_VEL
LIN {X 0,Y 566.478,Z 791.738,A -85,B 0,C 180,E1 25059.137,E2 25059.137} C_VEL
LIN {X 0,Y 570.12,Z 756.97,A -85,B 0,C 180,E1 25055.982,E2 25055.982} C_VEL
LIN {X 0,Y 573.674,Z 723.339,A -85,B 0,C 180,E1 25052.853,E2 25052.853} C_VEL
LIN {X 0,Y 575.329,Z 706.673,A -85,B 0,C 180,E1 25051.25,E2 25051.25} C_VEL
LIN {X 0,Y 567.44,Z 687.409,A -85,B 0,C 180,E1 25048.295,E2 25048.295} C_VEL
LIN {X 0,Y 559.754,Z 669.424,A -85,B 0,C 180,E1 25045.334,E2 25045.334} C_VEL
LIN {X 0,Y 552.186,Z 652.634,A -85,B 0,C 180,E1 25042.35,E2 25042.35} C_VEL
LIN {X 0,Y 545.541,Z 638.08,A -85,B 0,C 180,E1 25039.598,E2 25039.598} C_VEL
LIN {X 0,Y 541.117,Z 628.994,A -85,B 0,C 180,E1 25037.752,E2 25037.752} C_VEL
LIN {X 0,Y 539.24,Z 624.931,A -85,B 0,C 180,E1 25036.925,E2 25036.925} C_VEL
LIN {X 0,Y 537.684,Z 621.394,A -85,B 0,C 180,E1 25036.197,E2 25036.197} C_VEL
LIN {X 0,Y 537.625,Z 621.014,A -85,B 0,C 180,E1 25036.088,E2 25036.088} C_VEL
LIN {X 0,Y 537.612,Z 621.007,A -85,B 0,C 180,E1 25032.678,E2 25032.678} C_VEL
LIN {X 0,Y 537.611,Z 621.013,A -85,B 0,C 180,E1 25029.312,E2 25029.312} C_VEL
LIN {X 0,Y 537.616,Z 621.004,A -85,B 0,C 180,E1 25025.978,E2 25025.978} C_VEL
LIN {X 0,Y 537.622,Z 621.013,A -85,B 0,C 180,E1 25022.452,E2 25022.452} C_VEL
LIN {X 0,Y 537.629,Z 621.008,A -85,B 0,C 180,E1 25019.041,E2 25019.041} C_VEL
LIN {X 0,Y 537.628,Z 621.005,A -85,B 0,C 180,E1 25015.52,E2 25015.52} C_VEL
LIN {X 0,Y 537.623,Z 621.009,A -85,B 0,C 180,E1 25012.089,E2 25012.089} C_VEL
LIN {X 0,Y 537.612,Z 621.013,A -85,B 0,C 180,E1 25008.63,E2 25008.63} C_VEL
LIN {X 0,Y 537.613,Z 621.013,A -85,B 0,C 180,E1 25005.238,E2 25005.238} C_VEL
LIN {X 0,Y 537.624,Z 621.013,A -85,B 0,C 180,E1 25001.793,E2 25001.793} C_VEL
LIN {X 0,Y 537.633,Z 621.013,A -85,B 0,C 180,E1 24998.393,E2 24998.393} C_VEL
LIN {X 0,Y 537.63,Z 621.015,A -85,B 0,C 180,E1 24994.91,E2 24994.91} C_VEL
LIN {X 0,Y 537.629,Z 621.011,A -85,B 0,C 180,E1 24991.377,E2 24991.377} C_VEL
LIN {X 0,Y 537.617,Z 621.01,A -85,B 0,C 180,E1 24987.99,E2 24987.99} C_VEL
LIN {X 0,Y 537.611,Z 621.004,A -85,B 0,C 180,E1 24984.66,E2 24984.66} C_VEL
LIN {X 0,Y 537.614,Z 621.004,A -85,B 0,C 180,E1 24981.324,E2 24981.324} C_VEL
LIN {X 0,Y 537.623,Z 620.993,A -85,B 0,C 180,E1 24977.905,E2 24977.905} C_VEL
LIN {X 0,Y 537.627,Z 621.009,A -85,B 0,C 180,E1 24974.424,E2 24974.424} C_VEL
LIN {X 0,Y 537.612,Z 620.993,A -85,B 0,C 180,E1 24970.965,E2 24970.965} C_VEL
LIN {X 0,Y 537.627,Z 620.995,A -85,B 0,C 180,E1 24967.589,E2 24967.589} C_VEL
LIN {X 0,Y 537.629,Z 621.126,A -85,B 0,C 180,E1 24966.819,E2 24966.819} C_VEL
LIN {X 0,Y 546.478,Z 646.011,A -85,B 0,C 180,E1 24964.426,E2 24964.426} C_VEL
LIN {X 0,Y 552.273,Z 665.108,A -85,B 0,C 180,E1 24962.66,E2 24962.66} C_VEL
LIN {X 0,Y 550.7,Z 706.294,A -85,B 0,C 180,E1 24959.652,E2 24959.652} C_VEL
LIN {X 0,Y 548.676,Z 752.788,A -85,B 0,C 180,E1 24956.225,E2 24956.225} C_VEL
LIN {X 0,Y 546.784,Z 800.786,A -85,B 0,C 180,E1 24952.751,E2 24952.751} C_VEL
LIN {X 0,Y 545.485,Z 846.351,A -85,B 0,C 180,E1 24949.607,E2 24949.607} C_VEL
LIN {X 0,Y 546.275,Z 854.693,A -85,B 0,C 180,E1 24949.46,E2 24949.46} C_VEL
LIN {X 0,Y 545.779,Z 890.637,A -85,B 0,C 180,E1 24948.984,E2 24948.984} C_VEL
LIN {X 0,Y 544.785,Z 898.31,A -85,B 0,C 180,E1 24948.917,E2 24948.917} C_VEL
LIN {X 0,Y 538.598,Z 918.647,A -85,B 0,C 180,E1 24948.876,E2 24948.876} C_VEL
LIN {X 0,Y 537.817,Z 925.236,A -85,B 0,C 180,E1 24948.815,E2 24948.815} C_VEL
LIN {X 0,Y 536.755,Z 1017.576,A -85,B 0,C 180,E1 24947.542,E2 24947.542} C_VEL
LIN {X 0,Y 536.485,Z 1035.069,A -85,B 0,C 180,E1 24947.107,E2 24947.107} C_VEL
LIN {X 0,Y 535.936,Z 1052.106,A -85,B 0,C 180,E1 24946.47,E2 24946.47} C_VEL
LIN {X 0,Y 535.209,Z 1068.194,A -85,B 0,C 180,E1 24945.66,E2 24945.66} C_VEL
LIN {X 0,Y 534.347,Z 1083.311,A -85,B 0,C 180,E1 24944.686,E2 24944.686} C_VEL
LIN {X 0,Y 533.401,Z 1097.328,A -85,B 0,C 180,E1 24943.55,E2 24943.55} C_VEL
LIN {X 0,Y 532.428,Z 1110.307,A -85,B 0,C 180,E1 24942.25,E2 24942.25} C_VEL
LIN {X 0,Y 531.52,Z 1121.793,A -85,B 0,C 180,E1 24940.841,E2 24940.841} C_VEL
LIN {X 0,Y 530.717,Z 1131.867,A -85,B 0,C 180,E1 24939.323,E2 24939.323} C_VEL
LIN {X 0,Y 530.041,Z 1140.486,A -85,B 0,C 180,E1 24937.696,E2 24937.696} C_VEL
LIN {X 0,Y 529.518,Z 1147.671,A -85,B 0,C 180,E1 24935.96,E2 24935.96} C_VEL
LIN {X 0,Y 529.148,Z 1153.355,A -85,B 0,C 180,E1 24934.116,E2 24934.116} C_VEL
LIN {X 0,Y 528.93,Z 1157.227,A -85,B 0,C 180,E1 24932.274,E2 24932.274} C_VEL
LIN {X 0,Y 528.82,Z 1159.427,A -85,B 0,C 180,E1 24930.324,E2 24930.324} C_VEL
LIN {X 0,Y 528.799,Z 1159.838,A -85,B 0,C 180,E1 24928.373,E2 24928.373} C_VEL
LIN {X 0,Y 528.885,Z 1158.471,A -85,B 0,C 180,E1 24926.422,E2 24926.422} C_VEL
LIN {X 0,Y 529.065,Z 1155.424,A -85,B 0,C 180,E1 24924.576,E2 24924.576} C_VEL
LIN {X 0,Y 529.387,Z 1150.611,A -85,B 0,C 180,E1 24922.728,E2 24922.728} C_VEL
LIN {X 0,Y 529.879,Z 1143.902,A -85,B 0,C 180,E1 24920.878,E2 24920.878} C_VEL
LIN {X 0,Y 530.5,Z 1136.155,A -85,B 0,C 180,E1 24919.244,E2 24919.244} C_VEL
LIN {X 0,Y 531.311,Z 1126.312,A -85,B 0,C 180,E1 24917.61,E2 24917.61} C_VEL
LIN {X 0,Y 532.266,Z 1114.899,A -85,B 0,C 180,E1 24916.085,E2 24916.085} C_VEL
LIN {X 0,Y 533.27,Z 1102.35,A -85,B 0,C 180,E1 24914.724,E2 24914.724} C_VEL
LIN {X 0,Y 534.259,Z 1088.653,A -85,B 0,C 180,E1 24913.527,E2 24913.527} C_VEL
LIN {X 0,Y 535.178,Z 1073.974,A -85,B 0,C 180,E1 24912.493,E2 24912.493} C_VEL
LIN {X 0,Y 535.989,Z 1058.312,A -85,B 0,C 180,E1 24911.622,E2 24911.622} C_VEL
LIN {X 0,Y 536.613,Z 1042.207,A -85,B 0,C 180,E1 24910.939,E2 24910.939} C_VEL
LIN {X 0,Y 537.013,Z 1024.744,A -85,B 0,C 180,E1 24910.421,E2 24910.421} C_VEL
LIN {X 0,Y 537.162,Z 1005.14,A -85,B 0,C 180,E1 24910.068,E2 24910.068} C_VEL
LIN {X 0,Y 539.016,Z 852.024,A -85,B 0,C 180,E1 24907.994,E2 24907.994} C_VEL
LIN {X 0,Y 538.368,Z 846.983,A -85,B 0,C 180,E1 24907.878,E2 24907.878} C_VEL
LIN {X 0,Y 539.799,Z 801.721,A -85,B 0,C 180,E1 24904.718,E2 24904.718} C_VEL
LIN {X 0,Y 541.748,Z 756.141,A -85,B 0,C 180,E1 24901.382,E2 24901.382} C_VEL
LIN {X 0,Y 543.959,Z 708.573,A -85,B 0,C 180,E1 24897.848,E2 24897.848} C_VEL
LIN {X 0,Y 545.611,Z 668.26,A -85,B 0,C 180,E1 24894.869,E2 24894.869} C_VEL
LIN {X 0,Y 538.636,Z 646.292,A -85,B 0,C 180,E1 24892.758,E2 24892.758} C_VEL
LIN {X 0,Y 530.571,Z 624.756,A -85,B 0,C 180,E1 24890.594,E2 24890.594} C_VEL
LIN {X 0,Y 529.681,Z 621.973,A -85,B 0,C 180,E1 24890.317,E2 24890.317} C_VEL
LIN {X 0,Y 529.68,Z 621.996,A -85,B 0,C 180,E1 24886.892,E2 24886.892} C_VEL
LIN {X 0,Y 529.684,Z 622.003,A -85,B 0,C 180,E1 24883.383,E2 24883.383} C_VEL
LIN {X 0,Y 529.708,Z 622.218,A -85,B 0,C 180,E1 24882.432,E2 24882.432} C_VEL
LIN {X 0,Y 530.892,Z 625.329,A -85,B 0,C 180,E1 24881.93,E2 24881.93} C_VEL
LIN {X 0,Y 537.184,Z 638.451,A -85,B 0,C 180,E1 24879.779,E2 24879.779} C_VEL
LIN {X 0,Y 557.781,Z 668.287,A -85,B 0,C 180,E1 24877.32,E2 24877.32} C_VEL
LIN {X 0,Y 566.156,Z 681.034,A -85,B 0,C 180,E1 24876.37,E2 24876.37} C_VEL
LIN {X 0,Y 556.216,Z 923.957,A -85,B 0,C 180,E1 24872.457,E2 24872.457} C_VEL
LIN {X 0,Y 554.673,Z 967.613,A -85,B 0,C 180,E1 24871.723,E2 24871.723} C_VEL
LIN {X 0,Y 553.48,Z 990.428,A -85,B 0,C 180,E1 24871.147,E2 24871.147} C_VEL
LIN {X 0,Y 551.854,Z 1013.696,A -85,B 0,C 180,E1 24870.366,E2 24870.366} C_VEL
LIN {X 0,Y 549.981,Z 1035.536,A -85,B 0,C 180,E1 24869.442,E2 24869.442} C_VEL
LIN {X 0,Y 547.79,Z 1056.798,A -85,B 0,C 180,E1 24868.332,E2 24868.332} C_VEL
LIN {X 0,Y 545.446,Z 1077.438,A -85,B 0,C 180,E1 24867.041,E2 24867.041} C_VEL
LIN {X 0,Y 543.087,Z 1096.588,A -85,B 0,C 180,E1 24865.637,E2 24865.637} C_VEL
LIN {X 0,Y 540.567,Z 1115.279,A -85,B 0,C 180,E1 24864.013,E2 24864.013} C_VEL
LIN {X 0,Y 538.075,Z 1133.525,A -85,B 0,C 180,E1 24862.162,E2 24862.162} C_VEL
LIN {X 0,Y 535.906,Z 1149.331,A -85,B 0,C 180,E1 24860.306,E2 24860.306} C_VEL
LIN {X 0,Y 533.906,Z 1163.992,A -85,B 0,C 180,E1 24858.284,E2 24858.284} C_VEL
LIN {X 0,Y 532.114,Z 1177.962,A -85,B 0,C 180,E1 24856.035,E2 24856.035} C_VEL
LIN {X 0,Y 530.757,Z 1189.587,A -85,B 0,C 180,E1 24853.843,E2 24853.843} C_VEL
LIN {X 0,Y 529.683,Z 1199.738,A -85,B 0,C 180,E1 24851.543,E2 24851.543} C_VEL
LIN {X 0,Y 528.934,Z 1208.594,A -85,B 0,C 180,E1 24849.137,E2 24849.137} C_VEL
LIN {X 0,Y 528.47,Z 1215.339,A -85,B 0,C 180,E1 24846.846,E2 24846.846} C_VEL
LIN {X 0,Y 528.175,Z 1221.247,A -85,B 0,C 180,E1 24844.234,E2 24844.234} C_VEL
LIN {X 0,Y 528.06,Z 1224.942,A -85,B 0,C 180,E1 24841.953,E2 24841.953} C_VEL
LIN {X 0,Y 528.019,Z 1227.362,A -85,B 0,C 180,E1 24839.458,E2 24839.458} C_VEL
LIN {X 0,Y 528.004,Z 1228.249,A -85,B 0,C 180,E1 24837.178,E2 24837.178} C_VEL
LIN {X 0,Y 528.019,Z 1227.664,A -85,B 0,C 180,E1 24834.785,E2 24834.785} C_VEL
LIN {X 0,Y 528.072,Z 1225.709,A -85,B 0,C 180,E1 24832.383,E2 24832.383} C_VEL
LIN {X 0,Y 528.178,Z 1222.089,A -85,B 0,C 180,E1 24829.97,E2 24829.97} C_VEL
LIN {X 0,Y 528.441,Z 1216.912,A -85,B 0,C 180,E1 24827.517,E2 24827.517} C_VEL
LIN {X 0,Y 528.87,Z 1210.456,A -85,B 0,C 180,E1 24825.213,E2 24825.213} C_VEL
LIN {X 0,Y 529.606,Z 1201.826,A -85,B 0,C 180,E1 24822.758,E2 24822.758} C_VEL
LIN {X 0,Y 530.602,Z 1192.29,A -85,B 0,C 180,E1 24820.516,E2 24820.516} C_VEL
LIN {X 0,Y 531.84,Z 1181.308,A -85,B 0,C 180,E1 24818.377,E2 24818.377} C_VEL
LIN {X 0,Y 533.538,Z 1167.677,A -85,B 0,C 180,E1 24816.121,E2 24816.121} C_VEL
LIN {X 0,Y 535.317,Z 1154.085,A -85,B 0,C 180,E1 24814.199,E2 24814.199} C_VEL
LIN {X 0,Y 537.238,Z 1139.04,A -85,B 0,C 180,E1 24812.391,E2 24812.391} C_VEL
LIN {X 0,Y 539.324,Z 1122.718,A -85,B 0,C 180,E1 24810.696,E2 24810.696} C_VEL
LIN {X 0,Y 541.353,Z 1105.765,A -85,B 0,C 180,E1 24809.191,E2 24809.191} C_VEL
LIN {X 0,Y 543.321,Z 1087.479,A -85,B 0,C 180,E1 24807.813,E2 24807.813} C_VEL
LIN {X 0,Y 545.138,Z 1068.745,A -85,B 0,C 180,E1 24806.615,E2 24806.615} C_VEL
LIN {X 0,Y 546.59,Z 1050.357,A -85,B 0,C 180,E1 24805.643,E2 24805.643} C_VEL
LIN {X 0,Y 547.956,Z 1029.05,A -85,B 0,C 180,E1 24804.722,E2 24804.722} C_VEL
LIN {X 0,Y 548.907,Z 1007.858,A -85,B 0,C 180,E1 24804.005,E2 24804.005} C_VEL
LIN {X 0,Y 549.41,Z 986.388,A -85,B 0,C 180,E1 24803.483,E2 24803.483} C_VEL
LIN {X 0,Y 549.668,Z 958.403,A -85,B 0,C 180,E1 24803.042,E2 24803.042} C_VEL
LIN {X 0,Y 551.616,Z 866.496,A -85,B 0,C 180,E1 24801.741,E2 24801.741} C_VEL
LIN {X 0,Y 554.473,Z 785.835,A -85,B 0,C 180,E1 24800.436,E2 24800.436} C_VEL
LIN {X 0,Y 556.938,Z 733.64,A -85,B 0,C 180,E1 24799.494,E2 24799.494} C_VEL
LIN {X 0,Y 551.547,Z 736.193,A -85,B 0,C 180,E1 24798.953,E2 24798.953} C_VEL
LIN {X 0,Y 549.354,Z 736.909,A -85,B 0,C 180,E1 24798.7,E2 24798.7} C_VEL
LIN {X 0,Y 543.682,Z 742.067,A -85,B 0,C 180,E1 24798.068,E2 24798.068} C_VEL
LIN {X 0,Y 540.043,Z 744.36,A -85,B 0,C 180,E1 24797.548,E2 24797.548} C_VEL
LIN {X 0,Y 538.751,Z 744.877,A -85,B 0,C 180,E1 24797.304,E2 24797.304} C_VEL
LIN {X 0,Y 535.399,Z 763.205,A -85,B 0,C 180,E1 24795.514,E2 24795.514} C_VEL
LIN {X 0,Y 533.216,Z 785.226,A -85,B 0,C 180,E1 24793.57,E2 24793.57} C_VEL
LIN {X 0,Y 533.235,Z 806.297,A -85,B 0,C 180,E1 24791.809,E2 24791.809} C_VEL
LIN {X 0,Y 535.574,Z 826.959,A -85,B 0,C 180,E1 24790.127,E2 24790.127} C_VEL
LIN {X 0,Y 540.06,Z 846.037,A -85,B 0,C 180,E1 24788.605,E2 24788.605} C_VEL
LIN {X 0,Y 546.658,Z 864.043,A -85,B 0,C 180,E1 24787.196,E2 24787.196} C_VEL
LIN {X 0,Y 555.311,Z 881.307,A -85,B 0,C 180,E1 24785.877,E2 24785.877} C_VEL
LIN {X 0,Y 565.532,Z 897.138,A -85,B 0,C 180,E1 24784.722,E2 24784.722} C_VEL
LIN {X 0,Y 568.397,Z 901.292,A -85,B 0,C 180,E1 24784.477,E2 24784.477} C_VEL
LIN {X 0,Y 558.317,Z 930.345,A -85,B 0,C 180,E1 24784.594,E2 24784.594} C_VEL
LIN {X 0,Y 552.803,Z 950.35,A -85,B 0,C 180,E1 24784.546,E2 24784.546} C_VEL
LIN {X 0,Y 549.705,Z 966.528,A -85,B 0,C 180,E1 24784.357,E2 24784.357} C_VEL
LIN {X 0,Y 548.169,Z 982.497,A -85,B 0,C 180,E1 24784.024,E2 24784.024} C_VEL
LIN {X 0,Y 545.875,Z 1015.827,A -85,B 0,C 180,E1 24783.115,E2 24783.115} C_VEL
LIN {X 0,Y 543.595,Z 1047.309,A -85,B 0,C 180,E1 24782.052,E2 24782.052} C_VEL
LIN {X 0,Y 541.623,Z 1075.904,A -85,B 0,C 180,E1 24780.879,E2 24780.879} C_VEL
LIN {X 0,Y 539.8,Z 1102.619,A -85,B 0,C 180,E1 24779.582,E2 24779.582} C_VEL
LIN {X 0,Y 538.093,Z 1127.547,A -85,B 0,C 180,E1 24778.164,E2 24778.164} C_VEL
LIN {X 0,Y 536.44,Z 1151.631,A -85,B 0,C 180,E1 24776.575,E2 24776.575} C_VEL
LIN {X 0,Y 534.856,Z 1173.651,A -85,B 0,C 180,E1 24774.875,E2 24774.875} C_VEL
LIN {X 0,Y 533.421,Z 1193.272,A -85,B 0,C 180,E1 24773.124,E2 24773.124} C_VEL
LIN {X 0,Y 532.133,Z 1211.201,A -85,B 0,C 180,E1 24771.251,E2 24771.251} C_VEL
LIN {X 0,Y 531.031,Z 1226.821,A -85,B 0,C 180,E1 24769.355,E2 24769.355} C_VEL
LIN {X 0,Y 530.07,Z 1240.852,A -85,B 0,C 180,E1 24767.352,E2 24767.352} C_VEL
LIN {X 0,Y 529.314,Z 1253.398,A -85,B 0,C 180,E1 24765.224,E2 24765.224} C_VEL
LIN {X 0,Y 528.755,Z 1263.791,A -85,B 0,C 180,E1 24763.117,E2 24763.117} C_VEL
LIN {X 0,Y 528.379,Z 1272.625,A -85,B 0,C 180,E1 24760.91,E2 24760.91} C_VEL
LIN {X 0,Y 528.153,Z 1279.961,A -85,B 0,C 180,E1 24758.603,E2 24758.603} C_VEL
LIN {X 0,Y 528.048,Z 1285.386,A -85,B 0,C 180,E1 24756.307,E2 24756.307} C_VEL
LIN {X 0,Y 528,Z 1289.268,A -85,B 0,C 180,E1 24753.911,E2 24753.911} C_VEL
LIN {X 0,Y 527.991,Z 1291.28,A -85,B 0,C 180,E1 24751.629,E2 24751.629} C_VEL
LIN {X 0,Y 527.985,Z 1291.736,A -85,B 0,C 180,E1 24749.242,E2 24749.242} C_VEL
LIN {X 0,Y 527.98,Z 1290.602,A -85,B 0,C 180,E1 24746.962,E2 24746.962} C_VEL
LIN {X 0,Y 527.984,Z 1287.591,A -85,B 0,C 180,E1 24744.459,E2 24744.459} C_VEL
LIN {X 0,Y 528.041,Z 1283.238,A -85,B 0,C 180,E1 24742.166,E2 24742.166} C_VEL
LIN {X 0,Y 528.255,Z 1276.6,A -85,B 0,C 180,E1 24739.643,E2 24739.643} C_VEL
LIN {X 0,Y 528.619,Z 1268.765,A -85,B 0,C 180,E1 24737.327,E2 24737.327} C_VEL
LIN {X 0,Y 529.273,Z 1258.557,A -85,B 0,C 180,E1 24734.878,E2 24734.878} C_VEL
LIN {X 0,Y 530.198,Z 1246.846,A -85,B 0,C 180,E1 24732.553,E2 24732.553} C_VEL
LIN {X 0,Y 531.426,Z 1233.626,A -85,B 0,C 180,E1 24730.32,E2 24730.32} C_VEL
LIN {X 0,Y 533.147,Z 1217.266,A -85,B 0,C 180,E1 24727.972,E2 24727.972} C_VEL
LIN {X 0,Y 535.26,Z 1198.902,A -85,B 0,C 180,E1 24725.729,E2 24725.729} C_VEL
LIN {X 0,Y 537.576,Z 1179.802,A -85,B 0,C 180,E1 24723.727,E2 24723.727} C_VEL
LIN {X 0,Y 539.974,Z 1160.913,A -85,B 0,C 180,E1 24722.012,E2 24722.012} C_VEL
LIN {X 0,Y 542.39,Z 1141.935,A -85,B 0,C 180,E1 24720.516,E2 24720.516} C_VEL
LIN {X 0,Y 545.152,Z 1120.555,A -85,B 0,C 180,E1 24719.04,E2 24719.04} C_VEL
LIN {X 0,Y 547.841,Z 1099.26,A -85,B 0,C 180,E1 24717.798,E2 24717.798} C_VEL
LIN {X 0,Y 550.587,Z 1077.004,A -85,B 0,C 180,E1 24716.68,E2 24716.68} C_VEL
LIN {X 0,Y 553.313,Z 1053.409,A -85,B 0,C 180,E1 24715.714,E2 24715.714} C_VEL
LIN {X 0,Y 556.001,Z 1029.181,A -85,B 0,C 180,E1 24714.908,E2 24714.908} C_VEL
LIN {X 0,Y 558.238,Z 1004.695,A -85,B 0,C 180,E1 24714.295,E2 24714.295} C_VEL
LIN {X 0,Y 559.957,Z 977.499,A -85,B 0,C 180,E1 24713.779,E2 24713.779} C_VEL
LIN {X 0,Y 562.057,Z 959.529,A -85,B 0,C 180,E1 24713.572,E2 24713.572} C_VEL
LIN {X 0,Y 563.733,Z 949.777,A -85,B 0,C 180,E1 24713.478,E2 24713.478} C_VEL
LIN {X 0,Y 572.617,Z 935.016,A -85,B 0,C 180,E1 24712.707,E2 24712.707} C_VEL
LIN {X 0,Y 578.411,Z 925.72,A -85,B 0,C 180,E1 24712.241,E2 24712.241} C_VEL
LIN {X 0,Y 569.997,Z 913.482,A -85,B 0,C 180,E1 24710.679,E2 24710.679} C_VEL
LIN {X 0,Y 563.107,Z 899.38,A -85,B 0,C 180,E1 24708.996,E2 24708.996} C_VEL
LIN {X 0,Y 558.31,Z 884.44,A -85,B 0,C 180,E1 24707.322,E2 24707.322} C_VEL
LIN {X 0,Y 555.487,Z 868.134,A -85,B 0,C 180,E1 24705.612,E2 24705.612} C_VEL
LIN {X 0,Y 554.665,Z 849.677,A -85,B 0,C 180,E1 24703.808,E2 24703.808} C_VEL
LIN {X 0,Y 556.158,Z 827.089,A -85,B 0,C 180,E1 24701.749,E2 24701.749} C_VEL
LIN {X 0,Y 559.924,Z 791.382,A -85,B 0,C 180,E1 24698.544,E2 24698.544} C_VEL
LIN {X 0,Y 563.697,Z 756.939,A -85,B 0,C 180,E1 24695.385,E2 24695.385} C_VEL
LIN {X 0,Y 567.368,Z 723.92,A -85,B 0,C 180,E1 24692.275,E2 24692.275} C_VEL
LIN {X 0,Y 568.754,Z 710.694,A -85,B 0,C 180,E1 24691.005,E2 24691.005} C_VEL
LIN {X 0,Y 561.165,Z 692.08,A -85,B 0,C 180,E1 24688.12,E2 24688.12} C_VEL
LIN {X 0,Y 553.755,Z 674.608,A -85,B 0,C 180,E1 24685.223,E2 24685.223} C_VEL
LIN {X 0,Y 545.405,Z 655.783,A -85,B 0,C 180,E1 24681.849,E2 24681.849} C_VEL
LIN {X 0,Y 538.886,Z 642.024,A -85,B 0,C 180,E1 24679.173,E2 24679.173} C_VEL
LIN {X 0,Y 535.27,Z 634.318,A -85,B 0,C 180,E1 24677.615,E2 24677.615} C_VEL
LIN {X 0,Y 533.108,Z 629.853,A -85,B 0,C 180,E1 24676.676,E2 24676.676} C_VEL
LIN {X 0,Y 531.283,Z 625.904,A -85,B 0,C 180,E1 24675.837,E2 24675.837} C_VEL
LIN {X 0,Y 529.865,Z 622.958,A -85,B 0,C 180,E1 24675.207,E2 24675.207} C_VEL
LIN {X 0,Y 529.691,Z 621.993,A -85,B 0,C 180,E1 24674.988,E2 24674.988} C_VEL
LIN {X 0,Y 529.681,Z 621.999,A -85,B 0,C 180,E1 24671.543,E2 24671.543} C_VEL
LIN {X 0,Y 529.69,Z 621.995,A -85,B 0,C 180,E1 24668.03,E2 24668.03} C_VEL
LIN {X 0,Y 529.676,Z 622.001,A -85,B 0,C 180,E1 24664.439,E2 24664.439} C_VEL
LIN {X 0,Y 529.671,Z 621.994,A -85,B 0,C 180,E1 24660.973,E2 24660.973} C_VEL
LIN {X 0,Y 529.675,Z 621.999,A -85,B 0,C 180,E1 24657.62,E2 24657.62} C_VEL
LIN {X 0,Y 529.687,Z 622.004,A -85,B 0,C 180,E1 24654.141,E2 24654.141} C_VEL
LIN {X 0,Y 529.674,Z 622.001,A -85,B 0,C 180,E1 24650.766,E2 24650.766} C_VEL
LIN {X 0,Y 529.685,Z 621.997,A -85,B 0,C 180,E1 24647.351,E2 24647.351} C_VEL
LIN {X 0,Y 529.684,Z 621.996,A -85,B 0,C 180,E1 24643.889,E2 24643.889} C_VEL
LIN {X 0,Y 529.682,Z 621.996,A -85,B 0,C 180,E1 24640.366,E2 24640.366} C_VEL
LIN {X 0,Y 529.673,Z 621.998,A -85,B 0,C 180,E1 24636.998,E2 24636.998} C_VEL
LIN {X 0,Y 529.685,Z 621.995,A -85,B 0,C 180,E1 24633.545,E2 24633.545} C_VEL
LIN {X 0,Y 529.679,Z 621.998,A -85,B 0,C 180,E1 24630.108,E2 24630.108} C_VEL
LIN {X 0,Y 529.68,Z 622.001,A -85,B 0,C 180,E1 24626.743,E2 24626.743} C_VEL
LIN {X 0,Y 529.68,Z 622.002,A -85,B 0,C 180,E1 24623.244,E2 24623.244} C_VEL
LIN {X 0,Y 529.686,Z 622.002,A -85,B 0,C 180,E1 24619.693,E2 24619.693} C_VEL
LIN {X 0,Y 529.672,Z 621.967,A -85,B 0,C 180,E1 24616.297,E2 24616.297} C_VEL
LIN {X 0,Y 529.685,Z 621.991,A -85,B 0,C 180,E1 24612.909,E2 24612.909} C_VEL
LIN {X 0,Y 529.688,Z 622.009,A -85,B 0,C 180,E1 24609.46,E2 24609.46} C_VEL
LIN {X 0,Y 529.692,Z 622.063,A -85,B 0,C 180,E1 24607.294,E2 24607.294} C_VEL
LIN {X 0,Y 538.631,Z 646.87,A -85,B 0,C 180,E1 24604.864,E2 24604.864} C_VEL
LIN {X 0,Y 544.989,Z 667.444,A -85,B 0,C 180,E1 24602.922,E2 24602.922} C_VEL
LIN {X 0,Y 543.495,Z 705.167,A -85,B 0,C 180,E1 24600.147,E2 24600.147} C_VEL
LIN {X 0,Y 541.451,Z 751.523,A -85,B 0,C 180,E1 24596.72,E2 24596.72} C_VEL
LIN {X 0,Y 539.493,Z 798.313,A -85,B 0,C 180,E1 24593.308,E2 24593.308} C_VEL
LIN {X 0,Y 538.086,Z 843.316,A -85,B 0,C 180,E1 24590.162,E2 24590.162} C_VEL
LIN {X 0,Y 538.076,Z 847.737,A -85,B 0,C 180,E1 24589.891,E2 24589.891} C_VEL
LIN {X 0,Y 538.791,Z 855.589,A -85,B 0,C 180,E1 24589.751,E2 24589.751} C_VEL
LIN {X 0,Y 537.817,Z 925.236,A -85,B 0,C 180,E1 24588.815,E2 24588.815} C_VEL
LIN {X 0,Y 536.81,Z 932.907,A -85,B 0,C 180,E1 24588.747,E2 24588.747} C_VEL
LIN {X 0,Y 530.664,Z 953.247,A -85,B 0,C 180,E1 24588.703,E2 24588.703} C_VEL
LIN {X 0,Y 529.856,Z 959.835,A -85,B 0,C 180,E1 24588.641,E2 24588.641} C_VEL
LIN {X 0,Y 529.19,Z 1019.011,A -85,B 0,C 180,E1 24587.801,E2 24587.801} C_VEL
LIN {X 0,Y 528.898,Z 1036.445,A -85,B 0,C 180,E1 24587.354,E2 24587.354} C_VEL
LIN {X 0,Y 528.337,Z 1053.192,A -85,B 0,C 180,E1 24586.716,E2 24586.716} C_VEL
LIN {X 0,Y 527.588,Z 1069.135,A -85,B 0,C 180,E1 24585.902,E2 24585.902} C_VEL
LIN {X 0,Y 526.689,Z 1084.261,A -85,B 0,C 180,E1 24584.914,E2 24584.914} C_VEL
LIN {X 0,Y 525.694,Z 1098.377,A -85,B 0,C 180,E1 24583.752,E2 24583.752} C_VEL
LIN {X 0,Y 524.679,Z 1111.341,A -85,B 0,C 180,E1 24582.434,E2 24582.434} C_VEL
LIN {X 0,Y 523.728,Z 1122.815,A -85,B 0,C 180,E1 24581.005,E2 24581.005} C_VEL
LIN {X 0,Y 522.885,Z 1132.877,A -85,B 0,C 180,E1 24579.464,E2 24579.464} C_VEL
LIN {X 0,Y 522.173,Z 1141.482,A -85,B 0,C 180,E1 24577.812,E2 24577.812} C_VEL
LIN {X 0,Y 521.62,Z 1148.659,A -85,B 0,C 180,E1 24576.05,E2 24576.05} C_VEL
LIN {X 0,Y 521.228,Z 1154.334,A -85,B 0,C 180,E1 24574.179,E2 24574.179} C_VEL
LIN {X 0,Y 520.995,Z 1158.195,A -85,B 0,C 180,E1 24572.308,E2 24572.308} C_VEL
LIN {X 0,Y 520.877,Z 1160.385,A -85,B 0,C 180,E1 24570.328,E2 24570.328} C_VEL
LIN {X 0,Y 520.857,Z 1160.789,A -85,B 0,C 180,E1 24568.348,E2 24568.348} C_VEL
LIN {X 0,Y 520.95,Z 1159.413,A -85,B 0,C 180,E1 24566.367,E2 24566.367} C_VEL
LIN {X 0,Y 521.145,Z 1156.355,A -85,B 0,C 180,E1 24564.494,E2 24564.494} C_VEL
LIN {X 0,Y 521.49,Z 1151.533,A -85,B 0,C 180,E1 24562.618,E2 24562.618} C_VEL
LIN {X 0,Y 522.016,Z 1144.815,A -85,B 0,C 180,E1 24560.74,E2 24560.74} C_VEL
LIN {X 0,Y 522.677,Z 1137.053,A -85,B 0,C 180,E1 24559.082,E2 24559.082} C_VEL
LIN {X 0,Y 523.544,Z 1127.078,A -85,B 0,C 180,E1 24557.406,E2 24557.406} C_VEL
LIN {X 0,Y 524.539,Z 1115.766,A -85,B 0,C 180,E1 24555.876,E2 24555.876} C_VEL
LIN {X 0,Y 525.593,Z 1103.195,A -85,B 0,C 180,E1 24554.496,E2 24554.496} C_VEL
LIN {X 0,Y 526.614,Z 1089.678,A -85,B 0,C 180,E1 24553.298,E2 24553.298} C_VEL
LIN {X 0,Y 527.589,Z 1074.754,A -85,B 0,C 180,E1 24552.233,E2 24552.233} C_VEL
LIN {X 0,Y 528.434,Z 1059.046,A -85,B 0,C 180,E1 24551.349,E2 24551.349} C_VEL
LIN {X 0,Y 529.092,Z 1042.43,A -85,B 0,C 180,E1 24550.643,E2 24550.643} C_VEL
LIN {X 0,Y 529.497,Z 1025.054,A -85,B 0,C 180,E1 24550.127,E2 24550.127} C_VEL
LIN {X 0,Y 529.645,Z 1005.525,A -85,B 0,C 180,E1 24549.777,E2 24549.777} C_VEL
LIN {X 0,Y 531.59,Z 852.902,A -85,B 0,C 180,E1 24547.681,E2 24547.681} C_VEL
LIN {X 0,Y 530.953,Z 847.729,A -85,B 0,C 180,E1 24547.554,E2 24547.554} C_VEL
LIN {X 0,Y 532.432,Z 802.948,A -85,B 0,C 180,E1 24544.409,E2 24544.409} C_VEL
LIN {X 0,Y 534.48,Z 756.876,A -85,B 0,C 180,E1 24541.017,E2 24541.017} C_VEL
LIN {X 0,Y 536.707,Z 710.453,A -85,B 0,C 180,E1 24537.55,E2 24537.55} C_VEL
LIN {X 0,Y 538.421,Z 671.015,A -85,B 0,C 180,E1 24534.613,E2 24534.613} C_VEL
LIN {X 0,Y 531.65,Z 649.631,A -85,B 0,C 180,E1 24532.53,E2 24532.53} C_VEL
LIN {X 0,Y 523.536,Z 628.037,A -85,B 0,C 180,E1 24530.326,E2 24530.326} C_VEL
LIN {X 0,Y 521.733,Z 622.962,A -85,B 0,C 180,E1 24529.805,E2 24529.805} C_VEL
LIN {X 0,Y 521.744,Z 622.985,A -85,B 0,C 180,E1 24526.375,E2 24526.375} C_VEL
LIN {X 0,Y 521.746,Z 622.998,A -85,B 0,C 180,E1 24523.352,E2 24523.352} C_VEL
LIN {X 0,Y 523.077,Z 626.525,A -85,B 0,C 180,E1 24522.773,E2 24522.773} C_VEL
LIN {X 0,Y 527.782,Z 636.578,A -85,B 0,C 180,E1 24521.059,E2 24521.059} C_VEL
LIN {X 0,Y 529.76,Z 640.579,A -85,B 0,C 180,E1 24520.437,E2 24520.437} C_VEL
LIN {X 0,Y 549.179,Z 668.327,A -85,B 0,C 180,E1 24518.051,E2 24518.051} C_VEL
LIN {X 0,Y 559.74,Z 684.506,A -85,B 0,C 180,E1 24516.824,E2 24516.824} C_VEL
LIN {X 0,Y 549.103,Z 931.456,A -85,B 0,C 180,E1 24512.769,E2 24512.769} C_VEL
LIN {X 0,Y 547.69,Z 969.364,A -85,B 0,C 180,E1 24512.108,E2 24512.108} C_VEL
LIN {X 0,Y 546.46,Z 991.915,A -85,B 0,C 180,E1 24511.525,E2 24511.525} C_VEL
LIN {X 0,Y 544.785,Z 1014.819,A -85,B 0,C 180,E1 24510.741,E2 24510.741} C_VEL
LIN {X 0,Y 542.884,Z 1036.297,A -85,B 0,C 180,E1 24509.821,E2 24509.821} C_VEL
LIN {X 0,Y 540.688,Z 1056.792,A -85,B 0,C 180,E1 24508.739,E2 24508.739} C_VEL
LIN {X 0,Y 538.257,Z 1077.558,A -85,B 0,C 180,E1 24507.432,E2 24507.432} C_VEL
LIN {X 0,Y 535.805,Z 1096.741,A -85,B 0,C 180,E1 24506.011,E2 24506.011} C_VEL
LIN {X 0,Y 533.267,Z 1114.944,A -85,B 0,C 180,E1 24504.421,E2 24504.421} C_VEL
LIN {X 0,Y 530.741,Z 1132.873,A -85,B 0,C 180,E1 24502.602,E2 24502.602} C_VEL
LIN {X 0,Y 528.57,Z 1147.909,A -85,B 0,C 180,E1 24500.833,E2 24500.833} C_VEL
LIN {X 0,Y 526.502,Z 1162.532,A -85,B 0,C 180,E1 24498.836,E2 24498.836} C_VEL
LIN {X 0,Y 524.691,Z 1175.934,A -85,B 0,C 180,E1 24496.724,E2 24496.724} C_VEL
LIN {X 0,Y 523.183,Z 1187.826,A -85,B 0,C 180,E1 24494.499,E2 24494.499} C_VEL
LIN {X 0,Y 521.945,Z 1198.886,A -85,B 0,C 180,E1 24492.053,E2 24492.053} C_VEL
LIN {X 0,Y 521.13,Z 1207.638,A -85,B 0,C 180,E1 24489.721,E2 24489.721} C_VEL
LIN {X 0,Y 520.576,Z 1214.962,A -85,B 0,C 180,E1 24487.283,E2 24487.283} C_VEL
LIN {X 0,Y 520.26,Z 1220.751,A -85,B 0,C 180,E1 24484.851,E2 24484.851} C_VEL
LIN {X 0,Y 520.097,Z 1224.825,A -85,B 0,C 180,E1 24482.424,E2 24482.424} C_VEL
LIN {X 0,Y 520.039,Z 1227.589,A -85,B 0,C 180,E1 24479.89,E2 24479.89} C_VEL
LIN {X 0,Y 520.017,Z 1228.641,A -85,B 0,C 180,E1 24477.576,E2 24477.576} C_VEL
LIN {X 0,Y 520.031,Z 1228.318,A -85,B 0,C 180,E1 24475.036,E2 24475.036} C_VEL
LIN {X 0,Y 520.08,Z 1226.585,A -85,B 0,C 180,E1 24472.71,E2 24472.71} C_VEL
LIN {X 0,Y 520.192,Z 1223.091,A -85,B 0,C 180,E1 24470.15,E2 24470.15} C_VEL
LIN {X 0,Y 520.456,Z 1218.21,A -85,B 0,C 180,E1 24467.687,E2 24467.687} C_VEL
LIN {X 0,Y 520.894,Z 1211.83,A -85,B 0,C 180,E1 24465.322,E2 24465.322} C_VEL
LIN {X 0,Y 521.648,Z 1203.455,A -85,B 0,C 180,E1 24462.831,E2 24462.831} C_VEL
LIN {X 0,Y 522.662,Z 1194.085,A -85,B 0,C 180,E1 24460.557,E2 24460.557} C_VEL
LIN {X 0,Y 523.98,Z 1183.078,A -85,B 0,C 180,E1 24458.331,E2 24458.331} C_VEL
LIN {X 0,Y 525.615,Z 1170.791,A -85,B 0,C 180,E1 24456.21,E2 24456.21} C_VEL
LIN {X 0,Y 527.392,Z 1157.521,A -85,B 0,C 180,E1 24454.268,E2 24454.268} C_VEL
LIN {X 0,Y 529.518,Z 1142.042,A -85,B 0,C 180,E1 24452.321,E2 24452.321} C_VEL
LIN {X 0,Y 531.668,Z 1126.173,A -85,B 0,C 180,E1 24450.603,E2 24450.603} C_VEL
LIN {X 0,Y 533.789,Z 1109.273,A -85,B 0,C 180,E1 24449.056,E2 24449.056} C_VEL
LIN {X 0,Y 535.986,Z 1090.178,A -85,B 0,C 180,E1 24447.565,E2 24447.565} C_VEL
LIN {X 0,Y 537.871,Z 1071.904,A -85,B 0,C 180,E1 24446.36,E2 24446.36} C_VEL
LIN {X 0,Y 539.467,Z 1052.733,A -85,B 0,C 180,E1 24445.318,E2 24445.318} C_VEL
LIN {X 0,Y 540.898,Z 1031.764,A -85,B 0,C 180,E1 24444.387,E2 24444.387} C_VEL
LIN {X 0,Y 541.907,Z 1011.052,A -85,B 0,C 180,E1 24443.664,E2 24443.664} C_VEL
LIN {X 0,Y 542.456,Z 989.522,A -85,B 0,C 180,E1 24443.119,E2 24443.119} C_VEL
LIN {X 0,Y 542.729,Z 961.1,A -85,B 0,C 180,E1 24442.65,E2 24442.65} C_VEL
LIN {X 0,Y 544.797,Z 876.085,A -85,B 0,C 180,E1 24441.405,E2 24441.405} C_VEL
LIN {X 0,Y 547.861,Z 799.181,A -85,B 0,C 180,E1 24440.116,E2 24440.116} C_VEL
LIN {X 0,Y 550.829,Z 744.135,A -85,B 0,C 180,E1 24439.083,E2 24439.083} C_VEL
LIN {X 0,Y 543.93,Z 749.697,A -85,B 0,C 180,E1 24438.354,E2 24438.354} C_VEL
LIN {X 0,Y 539.571,Z 752.093,A -85,B 0,C 180,E1 24437.76,E2 24437.76} C_VEL
LIN {X 0,Y 532.909,Z 760.422,A -85,B 0,C 180,E1 24436.791,E2 24436.791} C_VEL
LIN {X 0,Y 528.741,Z 765.864,A -85,B 0,C 180,E1 24435.899,E2 24435.899} C_VEL
LIN {X 0,Y 528.011,Z 767.126,A -85,B 0,C 180,E1 24435.671,E2 24435.671} C_VEL
LIN {X 0,Y 525.734,Z 789.121,A -85,B 0,C 180,E1 24433.662,E2 24433.662} C_VEL
LIN {X 0,Y 525.771,Z 809.743,A -85,B 0,C 180,E1 24431.877,E2 24431.877} C_VEL
LIN {X 0,Y 528.235,Z 830.72,A -85,B 0,C 180,E1 24430.117,E2 24430.117} C_VEL
LIN {X 0,Y 532.759,Z 849.483,A -85,B 0,C 180,E1 24428.575,E2 24428.575} C_VEL
LIN {X 0,Y 536.036,Z 859.088,A -85,B 0,C 180,E1 24427.838,E2 24427.838} C_VEL
LIN {X 0,Y 543.889,Z 876.677,A -85,B 0,C 180,E1 24426.677,E2 24426.677} C_VEL
LIN {X 0,Y 553.944,Z 893.707,A -85,B 0,C 180,E1 24425.548,E2 24425.548} C_VEL
LIN {X 0,Y 560.476,Z 903.333,A -85,B 0,C 180,E1 24424.926,E2 24424.926} C_VEL
LIN {X 0,Y 551.797,Z 928.711,A -85,B 0,C 180,E1 24425.043,E2 24425.043} C_VEL
LIN {X 0,Y 546.046,Z 949.541,A -85,B 0,C 180,E1 24424.987,E2 24424.987} C_VEL
LIN {X 0,Y 542.795,Z 966.035,A -85,B 0,C 180,E1 24424.777,E2 24424.777} C_VEL
LIN {X 0,Y 541.127,Z 981.853,A -85,B 0,C 180,E1 24424.433,E2 24424.433} C_VEL
LIN {X 0,Y 538.561,Z 1016.334,A -85,B 0,C 180,E1 24423.454,E2 24423.454} C_VEL
LIN {X 0,Y 536.206,Z 1046.813,A -85,B 0,C 180,E1 24422.389,E2 24422.389} C_VEL
LIN {X 0,Y 533.988,Z 1076.808,A -85,B 0,C 180,E1 24421.12,E2 24421.12} C_VEL
LIN {X 0,Y 532,Z 1104.334,A -85,B 0,C 180,E1 24419.735,E2 24419.735} C_VEL
LIN {X 0,Y 530.186,Z 1129.538,A -85,B 0,C 180,E1 24418.254,E2 24418.254} C_VEL
LIN {X 0,Y 528.485,Z 1153.139,A -85,B 0,C 180,E1 24416.642,E2 24416.642} C_VEL
LIN {X 0,Y 526.882,Z 1174.993,A -85,B 0,C 180,E1 24414.918,E2 24414.918} C_VEL
LIN {X 0,Y 525.369,Z 1194.898,A -85,B 0,C 180,E1 24413.084,E2 24413.084} C_VEL
LIN {X 0,Y 524.085,Z 1212.564,A -85,B 0,C 180,E1 24411.196,E2 24411.196} C_VEL
LIN {X 0,Y 522.998,Z 1227.604,A -85,B 0,C 180,E1 24409.316,E2 24409.316} C_VEL
LIN {X 0,Y 522.031,Z 1241.592,A -85,B 0,C 180,E1 24407.272,E2 24407.272} C_VEL
LIN {X 0,Y 521.315,Z 1253.398,A -85,B 0,C 180,E1 24405.236,E2 24405.236} C_VEL
LIN {X 0,Y 520.752,Z 1263.708,A -85,B 0,C 180,E1 24403.097,E2 24403.097} C_VEL
LIN {X 0,Y 520.378,Z 1272.548,A -85,B 0,C 180,E1 24400.855,E2 24400.855} C_VEL
LIN {X 0,Y 520.161,Z 1279.534,A -85,B 0,C 180,E1 24398.625,E2 24398.625} C_VEL
LIN {X 0,Y 520.06,Z 1285.009,A -85,B 0,C 180,E1 24396.273,E2 24396.273} C_VEL
LIN {X 0,Y 520.015,Z 1288.718,A -85,B 0,C 180,E1 24393.971,E2 24393.971} C_VEL
LIN {X 0,Y 520.007,Z 1290.78,A -85,B 0,C 180,E1 24391.654,E2 24391.654} C_VEL
LIN {X 0,Y 519.999,Z 1291.26,A -85,B 0,C 180,E1 24389.23,E2 24389.23} C_VEL
LIN {X 0,Y 519.992,Z 1290.121,A -85,B 0,C 180,E1 24386.915,E2 24386.915} C_VEL
LIN {X 0,Y 519.993,Z 1287.253,A -85,B 0,C 180,E1 24384.484,E2 24384.484} C_VEL
LIN {X 0,Y 520.045,Z 1282.949,A -85,B 0,C 180,E1 24382.156,E2 24382.156} C_VEL
LIN {X 0,Y 520.247,Z 1276.646,A -85,B 0,C 180,E1 24379.705,E2 24379.705} C_VEL
LIN {X 0,Y 520.634,Z 1268.517,A -85,B 0,C 180,E1 24377.242,E2 24377.242} C_VEL
LIN {X 0,Y 521.312,Z 1258.259,A -85,B 0,C 180,E1 24374.747,E2 24374.747} C_VEL
LIN {X 0,Y 522.267,Z 1246.587,A -85,B 0,C 180,E1 24372.394,E2 24372.394} C_VEL
LIN {X 0,Y 523.546,Z 1233.363,A -85,B 0,C 180,E1 24370.128,E2 24370.128} C_VEL
LIN {X 0,Y 525.332,Z 1216.995,A -85,B 0,C 180,E1 24367.745,E2 24367.745} C_VEL
LIN {X 0,Y 527.4,Z 1199.693,A -85,B 0,C 180,E1 24365.59,E2 24365.59} C_VEL
LIN {X 0,Y 529.721,Z 1181.285,A -85,B 0,C 180,E1 24363.609,E2 24363.609} C_VEL
LIN {X 0,Y 532.431,Z 1160.747,A -85,B 0,C 180,E1 24361.702,E2 24361.702} C_VEL
LIN {X 0,Y 535.131,Z 1140.342,A -85,B 0,C 180,E1 24360.076,E2 24360.076} C_VEL
LIN {X 0,Y 538.039,Z 1118.87,A -85,B 0,C 180,E1 24358.584,E2 24358.584} C_VEL
LIN {X 0,Y 540.982,Z 1096.449,A -85,B 0,C 180,E1 24357.27,E2 24357.27} C_VEL
LIN {X 0,Y 543.857,Z 1074.057,A -85,B 0,C 180,E1 24356.149,E2 24356.149} C_VEL
LIN {X 0,Y 546.664,Z 1050.875,A -85,B 0,C 180,E1 24355.205,E2 24355.205} C_VEL
LIN {X 0,Y 549.428,Z 1026.616,A -85,B 0,C 180,E1 24354.402,E2 24354.402} C_VEL
LIN {X 0,Y 551.693,Z 1002.615,A -85,B 0,C 180,E1 24353.798,E2 24353.798} C_VEL
LIN {X 0,Y 553.727,Z 973.511,A -85,B 0,C 180,E1 24353.253,E2 24353.253} C_VEL
LIN {X 0,Y 556.653,Z 952.184,A -85,B 0,C 180,E1 24353.032,E2 24353.032} C_VEL
LIN {X 0,Y 557.386,Z 948.363,A -85,B 0,C 180,E1 24353,E2 24353} C_VEL
LIN {X 0,Y 566.362,Z 933.631,A -85,B 0,C 180,E1 24352.224,E2 24352.224} C_VEL
LIN {X 0,Y 569.945,Z 927.866,A -85,B 0,C 180,E1 24351.932,E2 24351.932} C_VEL
LIN {X 0,Y 561.495,Z 914.649,A -85,B 0,C 180,E1 24350.263,E2 24350.263} C_VEL
LIN {X 0,Y 555.005,Z 900.216,A -85,B 0,C 180,E1 24348.544,E2 24348.544} C_VEL
LIN {X 0,Y 550.422,Z 884.181,A -85,B 0,C 180,E1 24346.757,E2 24346.757} C_VEL
LIN {X 0,Y 548.043,Z 867.182,A -85,B 0,C 180,E1 24344.983,E2 24344.983} C_VEL
LIN {X 0,Y 547.756,Z 846.813,A -85,B 0,C 180,E1 24343.005,E2 24343.005} C_VEL
LIN {X 0,Y 552.798,Z 796.605,A -85,B 0,C 180,E1 24338.449,E2 24338.449} C_VEL
LIN {X 0,Y 556.71,Z 762.104,A -85,B 0,C 180,E1 24335.264,E2 24335.264} C_VEL
LIN {X 0,Y 560.549,Z 728.806,A -85,B 0,C 180,E1 24332.111,E2 24332.111} C_VEL
LIN {X 0,Y 562.055,Z 714.379,A -85,B 0,C 180,E1 24330.702,E2 24330.702} C_VEL
LIN {X 0,Y 554.119,Z 694.812,A -85,B 0,C 180,E1 24327.629,E2 24327.629} C_VEL
LIN {X 0,Y 546.119,Z 676.008,A -85,B 0,C 180,E1 24324.443,E2 24324.443} C_VEL
LIN {X 0,Y 537.791,Z 657.394,A -85,B 0,C 180,E1 24321.029,E2 24321.029} C_VEL
LIN {X 0,Y 531.363,Z 643.729,A -85,B 0,C 180,E1 24318.316,E2 24318.316} C_VEL
LIN {X 0,Y 527.283,Z 635.177,A -85,B 0,C 180,E1 24316.526,E2 24316.526} C_VEL
LIN {X 0,Y 525.406,Z 631.206,A -85,B 0,C 180,E1 24315.678,E2 24315.678} C_VEL
LIN {X 0,Y 523.306,Z 626.812,A -85,B 0,C 180,E1 24314.722,E2 24314.722} C_VEL
LIN {X 0,Y 521.809,Z 623.364,A -85,B 0,C 180,E1 24313.972,E2 24313.972} C_VEL
LIN {X 0,Y 521.749,Z 622.991,A -85,B 0,C 180,E1 24313.86,E2 24313.86} C_VEL
LIN {X 0,Y 521.734,Z 622.984,A -85,B 0,C 180,E1 24310.378,E2 24310.378} C_VEL
LIN {X 0,Y 521.75,Z 622.987,A -85,B 0,C 180,E1 24306.935,E2 24306.935} C_VEL
LIN {X 0,Y 521.738,Z 622.983,A -85,B 0,C 180,E1 24303.516,E2 24303.516} C_VEL
LIN {X 0,Y 521.737,Z 622.992,A -85,B 0,C 180,E1 24300.11,E2 24300.11} C_VEL
LIN {X 0,Y 521.736,Z 622.991,A -85,B 0,C 180,E1 24296.704,E2 24296.704} C_VEL
LIN {X 0,Y 521.754,Z 622.984,A -85,B 0,C 180,E1 24293.176,E2 24293.176} C_VEL
LIN {X 0,Y 521.739,Z 622.983,A -85,B 0,C 180,E1 24289.622,E2 24289.622} C_VEL
LIN {X 0,Y 521.753,Z 622.983,A -85,B 0,C 180,E1 24286.14,E2 24286.14} C_VEL
LIN {X 0,Y 521.74,Z 622.988,A -85,B 0,C 180,E1 24282.604,E2 24282.604} C_VEL
LIN {X 0,Y 521.734,Z 622.989,A -85,B 0,C 180,E1 24279.234,E2 24279.234} C_VEL
LIN {X 0,Y 521.739,Z 622.985,A -85,B 0,C 180,E1 24275.81,E2 24275.81} C_VEL
LIN {X 0,Y 521.755,Z 622.979,A -85,B 0,C 180,E1 24272.245,E2 24272.245} C_VEL
LIN {X 0,Y 521.749,Z 622.98,A -85,B 0,C 180,E1 24268.711,E2 24268.711} C_VEL
LIN {X 0,Y 521.745,Z 622.978,A -85,B 0,C 180,E1 24265.173,E2 24265.173} C_VEL
LIN {X 0,Y 521.738,Z 622.982,A -85,B 0,C 180,E1 24261.755,E2 24261.755} C_VEL
LIN {X 0,Y 521.734,Z 622.982,A -85,B 0,C 180,E1 24258.365,E2 24258.365} C_VEL
LIN {X 0,Y 521.744,Z 622.981,A -85,B 0,C 180,E1 24254.839,E2 24254.839} C_VEL
LIN {X 0,Y 521.749,Z 622.964,A -85,B 0,C 180,E1 24251.302,E2 24251.302} C_VEL
LIN {X 0,Y 521.764,Z 623.07,A -85,B 0,C 180,E1 24247.781,E2 24247.781} C_VEL
LIN {X 0,Y 530.925,Z 648.194,A -85,B 0,C 180,E1 24245.272,E2 24245.272} C_VEL
LIN {X 0,Y 537.68,Z 669.898,A -85,B 0,C 180,E1 24243.192,E2 24243.192} C_VEL
LIN {X 0,Y 536.216,Z 707.437,A -85,B 0,C 180,E1 24240.414,E2 24240.414} C_VEL
LIN {X 0,Y 534.041,Z 753.988,A -85,B 0,C 180,E1 24236.941,E2 24236.941} C_VEL
LIN {X 0,Y 531.991,Z 802.056,A -85,B 0,C 180,E1 24233.421,E2 24233.421} C_VEL
LIN {X 0,Y 530.558,Z 847.625,A -85,B 0,C 180,E1 24230.236,E2 24230.236} C_VEL
LIN {X 0,Y 531.326,Z 856.133,A -85,B 0,C 180,E1 24230.055,E2 24230.055} C_VEL
LIN {X 0,Y 529.856,Z 959.835,A -85,B 0,C 180,E1 24228.641,E2 24228.641} C_VEL
LIN {X 0,Y 528.811,Z 967.504,A -85,B 0,C 180,E1 24228.574,E2 24228.574} C_VEL
LIN {X 0,Y 522.662,Z 987.837,A -85,B 0,C 180,E1 24228.527,E2 24228.527} C_VEL
LIN {X 0,Y 521.845,Z 994.423,A -85,B 0,C 180,E1 24228.464,E2 24228.464} C_VEL
LIN {X 0,Y 521.625,Z 1022.17,A -85,B 0,C 180,E1 24228.032,E2 24228.032} C_VEL
LIN {X 0,Y 521.26,Z 1039.677,A -85,B 0,C 180,E1 24227.545,E2 24227.545} C_VEL
LIN {X 0,Y 520.642,Z 1056.776,A -85,B 0,C 180,E1 24226.856,E2 24226.856} C_VEL
LIN {X 0,Y 519.857,Z 1072.321,A -85,B 0,C 180,E1 24226.02,E2 24226.02} C_VEL
LIN {X 0,Y 518.867,Z 1087.605,A -85,B 0,C 180,E1 24224.963,E2 24224.963} C_VEL
LIN {X 0,Y 517.805,Z 1101.766,A -85,B 0,C 180,E1 24223.738,E2 24223.738} C_VEL
LIN {X 0,Y 516.775,Z 1114.327,A -85,B 0,C 180,E1 24222.4,E2 24222.4} C_VEL
LIN {X 0,Y 515.805,Z 1125.424,A -85,B 0,C 180,E1 24220.95,E2 24220.95} C_VEL
LIN {X 0,Y 514.885,Z 1135.728,A -85,B 0,C 180,E1 24219.274,E2 24219.274} C_VEL
LIN {X 0,Y 514.139,Z 1144.457,A -85,B 0,C 180,E1 24217.485,E2 24217.485} C_VEL
LIN {X 0,Y 513.614,Z 1151.189,A -85,B 0,C 180,E1 24215.696,E2 24215.696} C_VEL
LIN {X 0,Y 513.237,Z 1156.363,A -85,B 0,C 180,E1 24213.796,E2 24213.796} C_VEL
LIN {X 0,Y 513.007,Z 1159.932,A -85,B 0,C 180,E1 24211.786,E2 24211.786} C_VEL
LIN {X 0,Y 512.919,Z 1161.669,A -85,B 0,C 180,E1 24209.775,E2 24209.775} C_VEL
LIN {X 0,Y 512.931,Z 1161.531,A -85,B 0,C 180,E1 24207.764,E2 24207.764} C_VEL
LIN {X 0,Y 513.059,Z 1159.602,A -85,B 0,C 180,E1 24205.751,E2 24205.751} C_VEL
LIN {X 0,Y 513.318,Z 1156.068,A -85,B 0,C 180,E1 24203.848,E2 24203.848} C_VEL
LIN {X 0,Y 513.738,Z 1150.702,A -85,B 0,C 180,E1 24201.943,E2 24201.943} C_VEL
LIN {X 0,Y 514.32,Z 1143.808,A -85,B 0,C 180,E1 24200.148,E2 24200.148} C_VEL
LIN {X 0,Y 515.133,Z 1134.894,A -85,B 0,C 180,E1 24198.352,E2 24198.352} C_VEL
LIN {X 0,Y 516.05,Z 1125.097,A -85,B 0,C 180,E1 24196.782,E2 24196.782} C_VEL
LIN {X 0,Y 517.071,Z 1113.844,A -85,B 0,C 180,E1 24195.324,E2 24195.324} C_VEL
LIN {X 0,Y 518.196,Z 1100.593,A -85,B 0,C 180,E1 24193.93,E2 24193.93} C_VEL
LIN {X 0,Y 519.269,Z 1086.739,A -85,B 0,C 180,E1 24192.749,E2 24192.749} C_VEL
LIN {X 0,Y 520.241,Z 1072.013,A -85,B 0,C 180,E1 24191.742,E2 24191.742} C_VEL
LIN {X 0,Y 521.056,Z 1056.244,A -85,B 0,C 180,E1 24190.901,E2 24190.901} C_VEL
LIN {X 0,Y 521.698,Z 1038.872,A -85,B 0,C 180,E1 24190.209,E2 24190.209} C_VEL
LIN {X 0,Y 522.053,Z 1021.403,A -85,B 0,C 180,E1 24189.733,E2 24189.733} C_VEL
LIN {X 0,Y 522.416,Z 984.687,A -85,B 0,C 180,E1 24189.183,E2 24189.183} C_VEL
LIN {X 0,Y 524.198,Z 853.908,A -85,B 0,C 180,E1 24187.362,E2 24187.362} C_VEL
LIN {X 0,Y 523.559,Z 848.578,A -85,B 0,C 180,E1 24187.226,E2 24187.226} C_VEL
LIN {X 0,Y 525.094,Z 804.144,A -85,B 0,C 180,E1 24184.085,E2 24184.085} C_VEL
LIN {X 0,Y 527.123,Z 760.101,A -85,B 0,C 180,E1 24180.822,E2 24180.822} C_VEL
LIN {X 0,Y 529.487,Z 712.439,A -85,B 0,C 180,E1 24177.245,E2 24177.245} C_VEL
LIN {X 0,Y 531.255,Z 673.803,A -85,B 0,C 180,E1 24174.352,E2 24174.352} C_VEL
LIN {X 0,Y 524.404,Z 652.189,A -85,B 0,C 180,E1 24172.217,E2 24172.217} C_VEL
LIN {X 0,Y 516.432,Z 630.783,A -85,B 0,C 180,E1 24169.998,E2 24169.998} C_VEL
LIN {X 0,Y 513.816,Z 623.952,A -85,B 0,C 180,E1 24169.271,E2 24169.271} C_VEL
LIN {X 0,Y 513.797,Z 623.982,A -85,B 0,C 180,E1 24165.739,E2 24165.739} C_VEL
LIN {X 0,Y 513.817,Z 624.061,A -85,B 0,C 180,E1 24164.263,E2 24164.263} C_VEL
LIN {X 0,Y 514.96,Z 627.24,A -85,B 0,C 180,E1 24163.729,E2 24163.729} C_VEL
LIN {X 0,Y 516.124,Z 629.629,A -85,B 0,C 180,E1 24163.299,E2 24163.299} C_VEL
LIN {X 0,Y 521.797,Z 641.629,A -85,B 0,C 180,E1 24161.238,E2 24161.238} C_VEL
LIN {X 0,Y 523.09,Z 643.736,A -85,B 0,C 180,E1 24161.011,E2 24161.011} C_VEL
LIN {X 0,Y 538.082,Z 664.998,A -85,B 0,C 180,E1 24159.098,E2 24159.098} C_VEL
LIN {X 0,Y 553.329,Z 687.709,A -85,B 0,C 180,E1 24157.288,E2 24157.288} C_VEL
LIN {X 0,Y 542.085,Z 936.074,A -85,B 0,C 180,E1 24153.131,E2 24153.131} C_VEL
LIN {X 0,Y 540.7,Z 971.178,A -85,B 0,C 180,E1 24152.496,E2 24152.496} C_VEL
LIN {X 0,Y 539.424,Z 993.518,A -85,B 0,C 180,E1 24151.904,E2 24151.904} C_VEL
LIN {X 0,Y 537.727,Z 1015.777,A -85,B 0,C 180,E1 24151.127,E2 24151.127} C_VEL
LIN {X 0,Y 535.761,Z 1037.161,A -85,B 0,C 180,E1 24150.197,E2 24150.197} C_VEL
LIN {X 0,Y 533.389,Z 1058.597,A -85,B 0,C 180,E1 24149.047,E2 24149.047} C_VEL
LIN {X 0,Y 530.867,Z 1079.269,A -85,B 0,C 180,E1 24147.717,E2 24147.717} C_VEL
LIN {X 0,Y 528.357,Z 1098.254,A -85,B 0,C 180,E1 24146.285,E2 24146.285} C_VEL
LIN {X 0,Y 525.737,Z 1116.327,A -85,B 0,C 180,E1 24144.675,E2 24144.675} C_VEL
LIN {X 0,Y 523.05,Z 1134.624,A -85,B 0,C 180,E1 24142.775,E2 24142.775} C_VEL
LIN {X 0,Y 520.758,Z 1150.012,A -85,B 0,C 180,E1 24140.924,E2 24140.924} C_VEL
LIN {X 0,Y 518.635,Z 1164.404,A -85,B 0,C 180,E1 24138.899,E2 24138.899} C_VEL
LIN {X 0,Y 516.734,Z 1177.927,A -85,B 0,C 180,E1 24136.695,E2 24136.695} C_VEL
LIN {X 0,Y 515.243,Z 1189.374,A -85,B 0,C 180,E1 24134.498,E2 24134.498} C_VEL
LIN {X 0,Y 514.025,Z 1199.797,A -85,B 0,C 180,E1 24132.127,E2 24132.127} C_VEL
LIN {X 0,Y 513.183,Z 1208.515,A -85,B 0,C 180,E1 24129.759,E2 24129.759} C_VEL
LIN {X 0,Y 512.607,Z 1215.756,A -85,B 0,C 180,E1 24127.284,E2 24127.284} C_VEL
LIN {X 0,Y 512.277,Z 1221.455,A -85,B 0,C 180,E1 24124.815,E2 24124.815} C_VEL
LIN {X 0,Y 512.117,Z 1225.329,A -85,B 0,C 180,E1 24122.462,E2 24122.462} C_VEL
LIN {X 0,Y 512.054,Z 1228.085,A -85,B 0,C 180,E1 24119.888,E2 24119.888} C_VEL
LIN {X 0,Y 512.032,Z 1229.135,A -85,B 0,C 180,E1 24117.538,E2 24117.538} C_VEL
LIN {X 0,Y 512.049,Z 1228.79,A -85,B 0,C 180,E1 24114.959,E2 24114.959} C_VEL
LIN {X 0,Y 512.104,Z 1227.05,A -85,B 0,C 180,E1 24112.596,E2 24112.596} C_VEL
LIN {X 0,Y 512.232,Z 1223.528,A -85,B 0,C 180,E1 24109.995,E2 24109.995} C_VEL
LIN {X 0,Y 512.525,Z 1218.613,A -85,B 0,C 180,E1 24107.493,E2 24107.493} C_VEL
LIN {X 0,Y 513.006,Z 1212.218,A -85,B 0,C 180,E1 24105.091,E2 24105.091} C_VEL
LIN {X 0,Y 513.872,Z 1203.357,A -85,B 0,C 180,E1 24102.446,E2 24102.446} C_VEL
LIN {X 0,Y 514.992,Z 1193.923,A -85,B 0,C 180,E1 24100.137,E2 24100.137} C_VEL
LIN {X 0,Y 516.378,Z 1183.042,A -85,B 0,C 180,E1 24097.935,E2 24097.935} C_VEL
LIN {X 0,Y 518.161,Z 1170.276,A -85,B 0,C 180,E1 24095.731,E2 24095.731} C_VEL
LIN {X 0,Y 520.099,Z 1156.882,A -85,B 0,C 180,E1 24093.757,E2 24093.757} C_VEL
LIN {X 0,Y 522.21,Z 1142.121,A -85,B 0,C 180,E1 24091.899,E2 24091.899} C_VEL
LIN {X 0,Y 524.487,Z 1126.119,A -85,B 0,C 180,E1 24090.16,E2 24090.16} C_VEL
LIN {X 0,Y 526.704,Z 1109.328,A -85,B 0,C 180,E1 24088.609,E2 24088.609} C_VEL
LIN {X 0,Y 528.939,Z 1090.657,A -85,B 0,C 180,E1 24087.143,E2 24087.143} C_VEL
LIN {X 0,Y 530.91,Z 1072.284,A -85,B 0,C 180,E1 24085.923,E2 24085.923} C_VEL
LIN {X 0,Y 532.59,Z 1053.044,A -85,B 0,C 180,E1 24084.87,E2 24084.87} C_VEL
LIN {X 0,Y 534.022,Z 1032.482,A -85,B 0,C 180,E1 24083.957,E2 24083.957} C_VEL
LIN {X 0,Y 535.042,Z 1012.176,A -85,B 0,C 180,E1 24083.242,E2 24083.242} C_VEL
LIN {X 0,Y 535.607,Z 991.384,A -85,B 0,C 180,E1 24082.708,E2 24082.708} C_VEL
LIN {X 0,Y 535.921,Z 961.822,A -85,B 0,C 180,E1 24082.209,E2 24082.209} C_VEL
LIN {X 0,Y 538.225,Z 881.228,A -85,B 0,C 180,E1 24080.977,E2 24080.977} C_VEL
LIN {X 0,Y 541.562,Z 808.964,A -85,B 0,C 180,E1 24079.71,E2 24079.71} C_VEL
LIN {X 0,Y 544.772,Z 756.987,A -85,B 0,C 180,E1 24078.691,E2 24078.691} C_VEL
LIN {X 0,Y 539.928,Z 759.853,A -85,B 0,C 180,E1 24078.094,E2 24078.094} C_VEL
LIN {X 0,Y 533.344,Z 767.383,A -85,B 0,C 180,E1 24077.221,E2 24077.221} C_VEL
LIN {X 0,Y 528.375,Z 772.993,A -85,B 0,C 180,E1 24076.295,E2 24076.295} C_VEL
LIN {X 0,Y 523.219,Z 784.434,A -85,B 0,C 180,E1 24075.116,E2 24075.116} C_VEL
LIN {X 0,Y 520.281,Z 795.758,A -85,B 0,C 180,E1 24073.918,E2 24073.918} C_VEL
LIN {X 0,Y 519.327,Z 807.821,A -85,B 0,C 180,E1 24072.742,E2 24072.742} C_VEL
LIN {X 0,Y 520.211,Z 822.939,A -85,B 0,C 180,E1 24071.42,E2 24071.42} C_VEL
LIN {X 0,Y 523.249,Z 839.936,A -85,B 0,C 180,E1 24070.06,E2 24070.06} C_VEL
LIN {X 0,Y 528.577,Z 857.375,A -85,B 0,C 180,E1 24068.732,E2 24068.732} C_VEL
LIN {X 0,Y 536.818,Z 877.974,A -85,B 0,C 180,E1 24067.29,E2 24067.29} C_VEL
LIN {X 0,Y 545.842,Z 894.624,A -85,B 0,C 180,E1 24066.138,E2 24066.138} C_VEL
LIN {X 0,Y 552.785,Z 905.426,A -85,B 0,C 180,E1 24065.405,E2 24065.405} C_VEL
LIN {X 0,Y 545.845,Z 925.694,A -85,B 0,C 180,E1 24065.518,E2 24065.518} C_VEL
LIN {X 0,Y 539.765,Z 947.171,A -85,B 0,C 180,E1 24065.462,E2 24065.462} C_VEL
LIN {X 0,Y 536.355,Z 963.422,A -85,B 0,C 180,E1 24065.26,E2 24065.26} C_VEL
LIN {X 0,Y 534.347,Z 979.31,A -85,B 0,C 180,E1 24064.921,E2 24064.921} C_VEL
LIN {X 0,Y 531.554,Z 1014.25,A -85,B 0,C 180,E1 24063.901,E2 24063.901} C_VEL
LIN {X 0,Y 528.911,Z 1045.834,A -85,B 0,C 180,E1 24062.763,E2 24062.763} C_VEL
LIN {X 0,Y 526.554,Z 1075.403,A -85,B 0,C 180,E1 24061.482,E2 24061.482} C_VEL
LIN {X 0,Y 524.475,Z 1102.574,A -85,B 0,C 180,E1 24060.094,E2 24060.094} C_VEL
LIN {X 0,Y 522.49,Z 1128.914,A -85,B 0,C 180,E1 24058.521,E2 24058.521} C_VEL
LIN {X 0,Y 520.604,Z 1154.129,A -85,B 0,C 180,E1 24056.77,E2 24056.77} C_VEL
LIN {X 0,Y 518.909,Z 1176.361,A -85,B 0,C 180,E1 24054.962,E2 24054.962} C_VEL
LIN {X 0,Y 517.367,Z 1196.137,A -85,B 0,C 180,E1 24053.101,E2 24053.101} C_VEL
LIN {X 0,Y 516.06,Z 1213.61,A -85,B 0,C 180,E1 24051.175,E2 24051.175} C_VEL
LIN {X 0,Y 514.904,Z 1229.32,A -85,B 0,C 180,E1 24049.16,E2 24049.16} C_VEL
LIN {X 0,Y 513.997,Z 1242.359,A -85,B 0,C 180,E1 24047.2,E2 24047.2} C_VEL
LIN {X 0,Y 513.254,Z 1254.562,A -85,B 0,C 180,E1 24045.018,E2 24045.018} C_VEL
LIN {X 0,Y 512.69,Z 1264.868,A -85,B 0,C 180,E1 24042.801,E2 24042.801} C_VEL
LIN {X 0,Y 512.348,Z 1273.277,A -85,B 0,C 180,E1 24040.572,E2 24040.572} C_VEL
LIN {X 0,Y 512.136,Z 1280.366,A -85,B 0,C 180,E1 24038.163,E2 24038.163} C_VEL
LIN {X 0,Y 512.048,Z 1285.441,A -85,B 0,C 180,E1 24035.829,E2 24035.829} C_VEL
LIN {X 0,Y 512.028,Z 1288.805,A -85,B 0,C 180,E1 24033.472,E2 24033.472} C_VEL
LIN {X 0,Y 512.025,Z 1290.559,A -85,B 0,C 180,E1 24031.12,E2 24031.12} C_VEL
LIN {X 0,Y 512.013,Z 1290.674,A -85,B 0,C 180,E1 24028.771,E2 24028.771} C_VEL
LIN {X 0,Y 511.996,Z 1289.122,A -85,B 0,C 180,E1 24026.307,E2 24026.307} C_VEL
LIN {X 0,Y 512.009,Z 1286.049,A -85,B 0,C 180,E1 24023.948,E2 24023.948} C_VEL
LIN {X 0,Y 512.106,Z 1281.089,A -85,B 0,C 180,E1 24021.468,E2 24021.468} C_VEL
LIN {X 0,Y 512.334,Z 1274.466,A -85,B 0,C 180,E1 24019.015,E2 24019.015} C_VEL
LIN {X 0,Y 512.807,Z 1265.657,A -85,B 0,C 180,E1 24016.47,E2 24016.47} C_VEL
LIN {X 0,Y 513.542,Z 1255.451,A -85,B 0,C 180,E1 24014.068,E2 24014.068} C_VEL
LIN {X 0,Y 514.638,Z 1243.215,A -85,B 0,C 180,E1 24011.656,E2 24011.656} C_VEL
LIN {X 0,Y 516.144,Z 1228.647,A -85,B 0,C 180,E1 24009.238,E2 24009.238} C_VEL
LIN {X 0,Y 517.928,Z 1213.245,A -85,B 0,C 180,E1 24007.049,E2 24007.049} C_VEL
LIN {X 0,Y 520.181,Z 1195.425,A -85,B 0,C 180,E1 24004.864,E2 24004.864} C_VEL
LIN {X 0,Y 522.811,Z 1175.752,A -85,B 0,C 180,E1 24002.789,E2 24002.789} C_VEL
LIN {X 0,Y 525.527,Z 1155.743,A -85,B 0,C 180,E1 24000.978,E2 24000.978} C_VEL
LIN {X 0,Y 528.212,Z 1136.576,A -85,B 0,C 180,E1 23999.464,E2 23999.464} C_VEL
LIN {X 0,Y 531.43,Z 1113.47,A -85,B 0,C 180,E1 23997.894,E2 23997.894} C_VEL
LIN {X 0,Y 534.27,Z 1092.664,A -85,B 0,C 180,E1 23996.684,E2 23996.684} C_VEL
LIN {X 0,Y 537.526,Z 1068.206,A -85,B 0,C 180,E1 23995.493,E2 23995.493} C_VEL
LIN {X 0,Y 540.136,Z 1047.482,A -85,B 0,C 180,E1 23994.658,E2 23994.658} C_VEL
LIN {X 0,Y 543.125,Z 1021.509,A -85,B 0,C 180,E1 23993.818,E2 23993.818} C_VEL
LIN {X 0,Y 545.366,Z 998.265,A -85,B 0,C 180,E1 23993.239,E2 23993.239} C_VEL
LIN {X 0,Y 547.246,Z 972.547,A -85,B 0,C 180,E1 23992.765,E2 23992.765} C_VEL
LIN {X 0,Y 550.442,Z 950.428,A -85,B 0,C 180,E1 23992.531,E2 23992.531} C_VEL
LIN {X 0,Y 551.13,Z 946.837,A -85,B 0,C 180,E1 23992.506,E2 23992.506} C_VEL
LIN {X 0,Y 560.615,Z 931.455,A -85,B 0,C 180,E1 23991.699,E2 23991.699} C_VEL
LIN {X 0,Y 561.503,Z 929.842,A -85,B 0,C 180,E1 23991.61,E2 23991.61} C_VEL
LIN {X 0,Y 553.22,Z 916.015,A -85,B 0,C 180,E1 23989.866,E2 23989.866} C_VEL
LIN {X 0,Y 546.95,Z 900.901,A -85,B 0,C 180,E1 23988.078,E2 23988.078} C_VEL
LIN {X 0,Y 542.754,Z 884.377,A -85,B 0,C 180,E1 23986.234,E2 23986.234} C_VEL
LIN {X 0,Y 540.71,Z 866.188,A -85,B 0,C 180,E1 23984.347,E2 23984.347} C_VEL
LIN {X 0,Y 540.995,Z 844.878,A -85,B 0,C 180,E1 23982.281,E2 23982.281} C_VEL
LIN {X 0,Y 545.85,Z 800.257,A -85,B 0,C 180,E1 23978.205,E2 23978.205} C_VEL
LIN {X 0,Y 549.985,Z 764.995,A -85,B 0,C 180,E1 23974.926,E2 23974.926} C_VEL
LIN {X 0,Y 553.938,Z 731.933,A -85,B 0,C 180,E1 23971.773,E2 23971.773} C_VEL
LIN {X 0,Y 555.47,Z 718.351,A -85,B 0,C 180,E1 23970.435,E2 23970.435} C_VEL
LIN {X 0,Y 547.725,Z 699.162,A -85,B 0,C 180,E1 23967.389,E2 23967.389} C_VEL
LIN {X 0,Y 539.984,Z 680.902,A -85,B 0,C 180,E1 23964.273,E2 23964.273} C_VEL
LIN {X 0,Y 532.147,Z 663.354,A -85,B 0,C 180,E1 23961.032,E2 23961.032} C_VEL
LIN {X 0,Y 525.784,Z 649.513,A -85,B 0,C 180,E1 23958.287,E2 23958.287} C_VEL
LIN {X 0,Y 519.824,Z 636.916,A -85,B 0,C 180,E1 23955.622,E2 23955.622} C_VEL
LIN {X 0,Y 517.178,Z 631.7,A -85,B 0,C 180,E1 23954.442,E2 23954.442} C_VEL
LIN {X 0,Y 515.387,Z 627.843,A -85,B 0,C 180,E1 23953.577,E2 23953.577} C_VEL
LIN {X 0,Y 513.866,Z 624.4,A -85,B 0,C 180,E1 23952.816,E2 23952.816} C_VEL
LIN {X 0,Y 513.798,Z 623.972,A -85,B 0,C 180,E1 23952.704,E2 23952.704} C_VEL
LIN {X 0,Y 513.797,Z 623.977,A -85,B 0,C 180,E1 23949.182,E2 23949.182} C_VEL
LIN {X 0,Y 513.812,Z 623.97,A -85,B 0,C 180,E1 23945.696,E2 23945.696} C_VEL
LIN {X 0,Y 513.808,Z 623.979,A -85,B 0,C 180,E1 23942.119,E2 23942.119} C_VEL
LIN {X 0,Y 513.807,Z 623.971,A -85,B 0,C 180,E1 23938.662,E2 23938.662} C_VEL
LIN {X 0,Y 513.799,Z 623.975,A -85,B 0,C 180,E1 23935.088,E2 23935.088} C_VEL
LIN {X 0,Y 513.795,Z 623.979,A -85,B 0,C 180,E1 23931.72,E2 23931.72} C_VEL
LIN {X 0,Y 513.803,Z 623.98,A -85,B 0,C 180,E1 23928.188,E2 23928.188} C_VEL
LIN {X 0,Y 513.812,Z 623.98,A -85,B 0,C 180,E1 23924.653,E2 23924.653} C_VEL
LIN {X 0,Y 513.812,Z 623.978,A -85,B 0,C 180,E1 23921.153,E2 23921.153} C_VEL
LIN {X 0,Y 513.811,Z 623.977,A -85,B 0,C 180,E1 23917.566,E2 23917.566} C_VEL
LIN {X 0,Y 513.799,Z 623.98,A -85,B 0,C 180,E1 23914.032,E2 23914.032} C_VEL
LIN {X 0,Y 513.801,Z 623.981,A -85,B 0,C 180,E1 23910.632,E2 23910.632} C_VEL
LIN {X 0,Y 513.81,Z 623.982,A -85,B 0,C 180,E1 23907.116,E2 23907.116} C_VEL
LIN {X 0,Y 513.797,Z 623.982,A -85,B 0,C 180,E1 23903.59,E2 23903.59} C_VEL
LIN {X 0,Y 513.813,Z 623.978,A -85,B 0,C 180,E1 23900.058,E2 23900.058} C_VEL
LIN {X 0,Y 513.796,Z 623.941,A -85,B 0,C 180,E1 23896.54,E2 23896.54} C_VEL
LIN {X 0,Y 513.806,Z 623.971,A -85,B 0,C 180,E1 23893.081,E2 23893.081} C_VEL
LIN {X 0,Y 513.812,Z 623.984,A -85,B 0,C 180,E1 23889.59,E2 23889.59} C_VEL
LIN {X 0,Y 513.83,Z 624.13,A -85,B 0,C 180,E1 23888.285,E2 23888.285} C_VEL
LIN {X 0,Y 523.027,Z 648.937,A -85,B 0,C 180,E1 23885.754,E2 23885.754} C_VEL
LIN {X 0,Y 529.807,Z 670.299,A -85,B 0,C 180,E1 23883.665,E2 23883.665} C_VEL
LIN {X 0,Y 530.514,Z 673.319,A -85,B 0,C 180,E1 23883.389,E2 23883.389} C_VEL
LIN {X 0,Y 528.87,Z 710.299,A -85,B 0,C 180,E1 23880.63,E2 23880.63} C_VEL
LIN {X 0,Y 526.669,Z 756.634,A -85,B 0,C 180,E1 23877.165,E2 23877.165} C_VEL
LIN {X 0,Y 524.567,Z 804.324,A -85,B 0,C 180,E1 23873.654,E2 23873.654} C_VEL
LIN {X 0,Y 523.112,Z 849.095,A -85,B 0,C 180,E1 23870.511,E2 23870.511} C_VEL
LIN {X 0,Y 523.868,Z 857.171,A -85,B 0,C 180,E1 23870.361,E2 23870.361} C_VEL
LIN {X 0,Y 521.845,Z 994.423,A -85,B 0,C 180,E1 23868.464,E2 23868.464} C_VEL
LIN {X 0,Y 520.793,Z 1002.098,A -85,B 0,C 180,E1 23868.399,E2 23868.399} C_VEL
LIN {X 0,Y 514.983,Z 1021.339,A -85,B 0,C 180,E1 23868.316,E2 23868.316} C_VEL
LIN {X 0,Y 514.029,Z 1027.837,A -85,B 0,C 180,E1 23868.2,E2 23868.2} C_VEL
LIN {X 0,Y 513.997,Z 1028.922,A -85,B 0,C 180,E1 23868.175,E2 23868.175} C_VEL
LIN {X 0,Y 513.568,Z 1045.567,A -85,B 0,C 180,E1 23867.645,E2 23867.645} C_VEL
LIN {X 0,Y 512.89,Z 1061.34,A -85,B 0,C 180,E1 23866.943,E2 23866.943} C_VEL
LIN {X 0,Y 511.955,Z 1077.747,A -85,B 0,C 180,E1 23865.983,E2 23865.983} C_VEL
LIN {X 0,Y 510.956,Z 1092.202,A -85,B 0,C 180,E1 23864.91,E2 23864.91} C_VEL
LIN {X 0,Y 509.874,Z 1105.666,A -85,B 0,C 180,E1 23863.667,E2 23863.667} C_VEL
LIN {X 0,Y 508.774,Z 1118.085,A -85,B 0,C 180,E1 23862.253,E2 23862.253} C_VEL
LIN {X 0,Y 507.732,Z 1129.403,A -85,B 0,C 180,E1 23860.666,E2 23860.666} C_VEL
LIN {X 0,Y 506.836,Z 1139.153,A -85,B 0,C 180,E1 23858.965,E2 23858.965} C_VEL
LIN {X 0,Y 506.108,Z 1147.289,A -85,B 0,C 180,E1 23857.148,E2 23857.148} C_VEL
LIN {X 0,Y 505.577,Z 1153.867,A -85,B 0,C 180,E1 23855.218,E2 23855.218} C_VEL
LIN {X 0,Y 505.233,Z 1158.551,A -85,B 0,C 180,E1 23853.289,E2 23853.289} C_VEL
LIN {X 0,Y 505.028,Z 1161.552,A -85,B 0,C 180,E1 23851.246,E2 23851.246} C_VEL
LIN {X 0,Y 504.966,Z 1162.741,A -85,B 0,C 180,E1 23849.204,E2 23849.204} C_VEL
LIN {X 0,Y 505.02,Z 1162.154,A -85,B 0,C 180,E1 23847.161,E2 23847.161} C_VEL
LIN {X 0,Y 505.196,Z 1159.676,A -85,B 0,C 180,E1 23845.116,E2 23845.116} C_VEL
LIN {X 0,Y 505.545,Z 1155.298,A -85,B 0,C 180,E1 23843.069,E2 23843.069} C_VEL
LIN {X 0,Y 506.066,Z 1149.28,A -85,B 0,C 180,E1 23841.133,E2 23841.133} C_VEL
LIN {X 0,Y 506.778,Z 1141.526,A -85,B 0,C 180,E1 23839.289,E2 23839.289} C_VEL
LIN {X 0,Y 507.72,Z 1131.82,A -85,B 0,C 180,E1 23837.487,E2 23837.487} C_VEL
LIN {X 0,Y 508.774,Z 1121.074,A -85,B 0,C 180,E1 23835.894,E2 23835.894} C_VEL
LIN {X 0,Y 509.92,Z 1108.655,A -85,B 0,C 180,E1 23834.415,E2 23834.415} C_VEL
LIN {X 0,Y 511.12,Z 1094.613,A -85,B 0,C 180,E1 23833.063,E2 23833.063} C_VEL
LIN {X 0,Y 512.21,Z 1079.993,A -85,B 0,C 180,E1 23831.931,E2 23831.931} C_VEL
LIN {X 0,Y 513.137,Z 1064.855,A -85,B 0,C 180,E1 23831.008,E2 23831.008} C_VEL
LIN {X 0,Y 513.923,Z 1047.758,A -85,B 0,C 180,E1 23830.211,E2 23830.211} C_VEL
LIN {X 0,Y 514.433,Z 1030.415,A -85,B 0,C 180,E1 23829.631,E2 23829.631} C_VEL
LIN {X 0,Y 514.623,Z 1012.203,A -85,B 0,C 180,E1 23829.255,E2 23829.255} C_VEL
LIN {X 0,Y 516.805,Z 854.781,A -85,B 0,C 180,E1 23827.031,E2 23827.031} C_VEL
LIN {X 0,Y 516.179,Z 849.41,A -85,B 0,C 180,E1 23826.887,E2 23826.887} C_VEL
LIN {X 0,Y 517.766,Z 805.307,A -85,B 0,C 180,E1 23823.752,E2 23823.752} C_VEL
LIN {X 0,Y 519.965,Z 759.26,A -85,B 0,C 180,E1 23820.324,E2 23820.324} C_VEL
LIN {X 0,Y 522.402,Z 712.242,A -85,B 0,C 180,E1 23816.765,E2 23816.765} C_VEL
LIN {X 0,Y 524.083,Z 676.502,A -85,B 0,C 180,E1 23814.071,E2 23814.071} C_VEL
LIN {X 0,Y 517.199,Z 654.797,A -85,B 0,C 180,E1 23811.892,E2 23811.892} C_VEL
LIN {X 0,Y 509.59,Z 634.548,A -85,B 0,C 180,E1 23809.754,E2 23809.754} C_VEL
LIN {X 0,Y 505.871,Z 624.952,A -85,B 0,C 180,E1 23808.686,E2 23808.686} C_VEL
LIN {X 0,Y 505.874,Z 625.031,A -85,B 0,C 180,E1 23805.235,E2 23805.235} C_VEL
LIN {X 0,Y 507.201,Z 628.497,A -85,B 0,C 180,E1 23804.628,E2 23804.628} C_VEL
LIN {X 0,Y 508.176,Z 630.473,A -85,B 0,C 180,E1 23804.256,E2 23804.256} C_VEL
LIN {X 0,Y 514.633,Z 644.188,A -85,B 0,C 180,E1 23801.835,E2 23801.835} C_VEL
LIN {X 0,Y 531.6,Z 668.258,A -85,B 0,C 180,E1 23799.624,E2 23799.624} C_VEL
LIN {X 0,Y 546.942,Z 690.976,A -85,B 0,C 180,E1 23797.76,E2 23797.76} C_VEL
LIN {X 0,Y 534.938,Z 943.743,A -85,B 0,C 180,E1 23793.446,E2 23793.446} C_VEL
LIN {X 0,Y 533.641,Z 974.446,A -85,B 0,C 180,E1 23792.854,E2 23792.854} C_VEL
LIN {X 0,Y 532.275,Z 997.08,A -85,B 0,C 180,E1 23792.231,E2 23792.231} C_VEL
LIN {X 0,Y 530.502,Z 1018.685,A -85,B 0,C 180,E1 23791.441,E2 23791.441} C_VEL
LIN {X 0,Y 528.279,Z 1041.204,A -85,B 0,C 180,E1 23790.418,E2 23790.418} C_VEL
LIN {X 0,Y 525.997,Z 1061.291,A -85,B 0,C 180,E1 23789.307,E2 23789.307} C_VEL
LIN {X 0,Y 523.407,Z 1081.475,A -85,B 0,C 180,E1 23787.969,E2 23787.969} C_VEL
LIN {X 0,Y 520.701,Z 1100.925,A -85,B 0,C 180,E1 23786.456,E2 23786.456} C_VEL
LIN {X 0,Y 518.04,Z 1118.81,A -85,B 0,C 180,E1 23784.822,E2 23784.822} C_VEL
LIN {X 0,Y 515.465,Z 1135.639,A -85,B 0,C 180,E1 23783.033,E2 23783.033} C_VEL
LIN {X 0,Y 513.072,Z 1151.184,A -85,B 0,C 180,E1 23781.133,E2 23781.133} C_VEL
LIN {X 0,Y 510.874,Z 1165.486,A -85,B 0,C 180,E1 23779.078,E2 23779.078} C_VEL
LIN {X 0,Y 508.866,Z 1179.211,A -85,B 0,C 180,E1 23776.789,E2 23776.789} C_VEL
LIN {X 0,Y 507.299,Z 1190.9,A -85,B 0,C 180,E1 23774.496,E2 23774.496} C_VEL
LIN {X 0,Y 506.052,Z 1201.142,A -85,B 0,C 180,E1 23772.09,E2 23772.09} C_VEL
LIN {X 0,Y 505.198,Z 1209.713,A -85,B 0,C 180,E1 23769.685,E2 23769.685} C_VEL
LIN {X 0,Y 504.616,Z 1216.828,A -85,B 0,C 180,E1 23767.171,E2 23767.171} C_VEL
LIN {X 0,Y 504.269,Z 1222.553,A -85,B 0,C 180,E1 23764.549,E2 23764.549} C_VEL
LIN {X 0,Y 504.121,Z 1226.3,A -85,B 0,C 180,E1 23762.16,E2 23762.16} C_VEL
LIN {X 0,Y 504.065,Z 1228.787,A -85,B 0,C 180,E1 23759.545,E2 23759.545} C_VEL
LIN {X 0,Y 504.048,Z 1229.709,A -85,B 0,C 180,E1 23757.157,E2 23757.157} C_VEL
LIN {X 0,Y 504.073,Z 1229.15,A -85,B 0,C 180,E1 23754.651,E2 23754.651} C_VEL
LIN {X 0,Y 504.148,Z 1227.206,A -85,B 0,C 180,E1 23752.134,E2 23752.134} C_VEL
LIN {X 0,Y 504.298,Z 1223.598,A -85,B 0,C 180,E1 23749.605,E2 23749.605} C_VEL
LIN {X 0,Y 504.653,Z 1218.181,A -85,B 0,C 180,E1 23746.946,E2 23746.946} C_VEL
LIN {X 0,Y 505.229,Z 1211.638,A -85,B 0,C 180,E1 23744.504,E2 23744.504} C_VEL
LIN {X 0,Y 506.119,Z 1203.3,A -85,B 0,C 180,E1 23742.049,E2 23742.049} C_VEL
LIN {X 0,Y 507.336,Z 1193.717,A -85,B 0,C 180,E1 23739.704,E2 23739.704} C_VEL
LIN {X 0,Y 508.87,Z 1182.645,A -85,B 0,C 180,E1 23737.447,E2 23737.447} C_VEL
LIN {X 0,Y 510.765,Z 1169.799,A -85,B 0,C 180,E1 23735.233,E2 23735.233} C_VEL
LIN {X 0,Y 512.86,Z 1156.284,A -85,B 0,C 180,E1 23733.233,E2 23733.233} C_VEL
LIN {X 0,Y 515.025,Z 1141.799,A -85,B 0,C 180,E1 23731.408,E2 23731.408} C_VEL
LIN {X 0,Y 517.521,Z 1124.971,A -85,B 0,C 180,E1 23729.589,E2 23729.589} C_VEL
LIN {X 0,Y 519.888,Z 1107.966,A -85,B 0,C 180,E1 23728.014,E2 23728.014} C_VEL
LIN {X 0,Y 522.104,Z 1089.986,A -85,B 0,C 180,E1 23726.616,E2 23726.616} C_VEL
LIN {X 0,Y 524.199,Z 1070.812,A -85,B 0,C 180,E1 23725.359,E2 23725.359} C_VEL
LIN {X 0,Y 525.986,Z 1051.287,A -85,B 0,C 180,E1 23724.296,E2 23724.296} C_VEL
LIN {X 0,Y 527.363,Z 1031.336,A -85,B 0,C 180,E1 23723.428,E2 23723.428} C_VEL
LIN {X 0,Y 528.371,Z 1009.733,A -85,B 0,C 180,E1 23722.696,E2 23722.696} C_VEL
LIN {X 0,Y 528.922,Z 988.916,A -85,B 0,C 180,E1 23722.182,E2 23722.182} C_VEL
LIN {X 0,Y 529.749,Z 943.057,A -85,B 0,C 180,E1 23721.446,E2 23721.446} C_VEL
LIN {X 0,Y 532.509,Z 870.807,A -85,B 0,C 180,E1 23720.247,E2 23720.247} C_VEL
LIN {X 0,Y 536.485,Z 803.132,A -85,B 0,C 180,E1 23718.969,E2 23718.969} C_VEL
LIN {X 0,Y 538.983,Z 769.239,A -85,B 0,C 180,E1 23718.266,E2 23718.266} C_VEL
LIN {X 0,Y 531.973,Z 776.429,A -85,B 0,C 180,E1 23717.341,E2 23717.341} C_VEL
LIN {X 0,Y 528.318,Z 780.337,A -85,B 0,C 180,E1 23716.715,E2 23716.715} C_VEL
LIN {X 0,Y 522.408,Z 791.767,A -85,B 0,C 180,E1 23715.556,E2 23715.556} C_VEL
LIN {X 0,Y 518.69,Z 802.998,A -85,B 0,C 180,E1 23714.367,E2 23714.367} C_VEL
LIN {X 0,Y 516.935,Z 815.116,A -85,B 0,C 180,E1 23713.166,E2 23713.166} C_VEL
LIN {X 0,Y 517.036,Z 829.461,A -85,B 0,C 180,E1 23711.879,E2 23711.879} C_VEL
LIN {X 0,Y 519.337,Z 845.663,A -85,B 0,C 180,E1 23710.526,E2 23710.526} C_VEL
LIN {X 0,Y 523.971,Z 862.539,A -85,B 0,C 180,E1 23709.173,E2 23709.173} C_VEL
LIN {X 0,Y 531.368,Z 882.187,A -85,B 0,C 180,E1 23707.735,E2 23707.735} C_VEL
LIN {X 0,Y 540.032,Z 898.894,A -85,B 0,C 180,E1 23706.527,E2 23706.527} C_VEL
LIN {X 0,Y 545.199,Z 907.3,A -85,B 0,C 180,E1 23705.932,E2 23705.932} C_VEL
LIN {X 0,Y 538.791,Z 926.846,A -85,B 0,C 180,E1 23706.024,E2 23706.024} C_VEL
LIN {X 0,Y 533.114,Z 946.961,A -85,B 0,C 180,E1 23705.949,E2 23705.949} C_VEL
LIN {X 0,Y 529.505,Z 964.229,A -85,B 0,C 180,E1 23705.716,E2 23705.716} C_VEL
LIN {X 0,Y 527.38,Z 980.8,A -85,B 0,C 180,E1 23705.33,E2 23705.33} C_VEL
LIN {X 0,Y 524.268,Z 1016.051,A -85,B 0,C 180,E1 23704.239,E2 23704.239} C_VEL
LIN {X 0,Y 521.466,Z 1047.375,A -85,B 0,C 180,E1 23703.061,E2 23703.061} C_VEL
LIN {X 0,Y 518.976,Z 1076.837,A -85,B 0,C 180,E1 23701.735,E2 23701.735} C_VEL
LIN {X 0,Y 516.713,Z 1104.842,A -85,B 0,C 180,E1 23700.253,E2 23700.253} C_VEL
LIN {X 0,Y 514.68,Z 1130.361,A -85,B 0,C 180,E1 23698.677,E2 23698.677} C_VEL
LIN {X 0,Y 512.856,Z 1153.63,A -85,B 0,C 180,E1 23697.019,E2 23697.019} C_VEL
LIN {X 0,Y 511.093,Z 1175.922,A -85,B 0,C 180,E1 23695.184,E2 23695.184} C_VEL
LIN {X 0,Y 509.547,Z 1195.129,A -85,B 0,C 180,E1 23693.354,E2 23693.354} C_VEL
LIN {X 0,Y 508.155,Z 1213.178,A -85,B 0,C 180,E1 23691.349,E2 23691.349} C_VEL
LIN {X 0,Y 506.994,Z 1228.619,A -85,B 0,C 180,E1 23689.351,E2 23689.351} C_VEL
LIN {X 0,Y 506.052,Z 1241.707,A -85,B 0,C 180,E1 23687.36,E2 23687.36} C_VEL
LIN {X 0,Y 505.285,Z 1254.032,A -85,B 0,C 180,E1 23685.143,E2 23685.143} C_VEL
LIN {X 0,Y 504.711,Z 1264.337,A -85,B 0,C 180,E1 23682.912,E2 23682.912} C_VEL
LIN {X 0,Y 504.371,Z 1272.477,A -85,B 0,C 180,E1 23680.741,E2 23680.741} C_VEL
LIN {X 0,Y 504.161,Z 1279.602,A -85,B 0,C 180,E1 23678.326,E2 23678.326} C_VEL
LIN {X 0,Y 504.071,Z 1284.649,A -85,B 0,C 180,E1 23676.036,E2 23676.036} C_VEL
LIN {X 0,Y 504.04,Z 1288.148,A -85,B 0,C 180,E1 23673.641,E2 23673.641} C_VEL
LIN {X 0,Y 504.037,Z 1290.006,A -85,B 0,C 180,E1 23671.252,E2 23671.252} C_VEL
LIN {X 0,Y 504.032,Z 1290.255,A -85,B 0,C 180,E1 23668.953,E2 23668.953} C_VEL
LIN {X 0,Y 504.011,Z 1288.831,A -85,B 0,C 180,E1 23666.476,E2 23666.476} C_VEL
LIN {X 0,Y 504.017,Z 1285.714,A -85,B 0,C 180,E1 23663.966,E2 23663.966} C_VEL
LIN {X 0,Y 504.111,Z 1280.768,A -85,B 0,C 180,E1 23661.447,E2 23661.447} C_VEL
LIN {X 0,Y 504.346,Z 1274.049,A -85,B 0,C 180,E1 23658.914,E2 23658.914} C_VEL
LIN {X 0,Y 504.83,Z 1265.354,A -85,B 0,C 180,E1 23656.369,E2 23656.369} C_VEL
LIN {X 0,Y 505.589,Z 1255.143,A -85,B 0,C 180,E1 23653.928,E2 23653.928} C_VEL
LIN {X 0,Y 506.797,Z 1242.252,A -85,B 0,C 180,E1 23651.362,E2 23651.362} C_VEL
LIN {X 0,Y 508.379,Z 1227.557,A -85,B 0,C 180,E1 23648.906,E2 23648.906} C_VEL
LIN {X 0,Y 510.253,Z 1212.036,A -85,B 0,C 180,E1 23646.684,E2 23646.684} C_VEL
LIN {X 0,Y 512.544,Z 1194.59,A -85,B 0,C 180,E1 23644.524,E2 23644.524} C_VEL
LIN {X 0,Y 515.364,Z 1174.38,A -85,B 0,C 180,E1 23642.376,E2 23642.376} C_VEL
LIN {X 0,Y 518.223,Z 1154.091,A -85,B 0,C 180,E1 23640.529,E2 23640.529} C_VEL
LIN {X 0,Y 521.175,Z 1133.979,A -85,B 0,C 180,E1 23638.932,E2 23638.932} C_VEL
LIN {X 0,Y 524.391,Z 1111.616,A -85,B 0,C 180,E1 23637.41,E2 23637.41} C_VEL
LIN {X 0,Y 527.582,Z 1089.332,A -85,B 0,C 180,E1 23636.111,E2 23636.111} C_VEL
LIN {X 0,Y 530.749,Z 1066.351,A -85,B 0,C 180,E1 23634.997,E2 23634.997} C_VEL
LIN {X 0,Y 533.535,Z 1044.956,A -85,B 0,C 180,E1 23634.131,E2 23634.131} C_VEL
LIN {X 0,Y 536.625,Z 1019.027,A -85,B 0,C 180,E1 23633.295,E2 23633.295} C_VEL
LIN {X 0,Y 539.072,Z 994.034,A -85,B 0,C 180,E1 23632.672,E2 23632.672} C_VEL
LIN {X 0,Y 540.869,Z 971.05,A -85,B 0,C 180,E1 23632.258,E2 23632.258} C_VEL
LIN {X 0,Y 544.404,Z 947.675,A -85,B 0,C 180,E1 23632.022,E2 23632.022} C_VEL
LIN {X 0,Y 544.894,Z 945.33,A -85,B 0,C 180,E1 23632.003,E2 23632.003} C_VEL
LIN {X 0,Y 553.168,Z 931.836,A -85,B 0,C 180,E1 23631.29,E2 23631.29} C_VEL
LIN {X 0,Y 545.234,Z 917.785,A -85,B 0,C 180,E1 23629.522,E2 23629.522} C_VEL
LIN {X 0,Y 539.262,Z 902.418,A -85,B 0,C 180,E1 23627.698,E2 23627.698} C_VEL
LIN {X 0,Y 535.319,Z 885.635,A -85,B 0,C 180,E1 23625.828,E2 23625.828} C_VEL
LIN {X 0,Y 533.567,Z 867.157,A -85,B 0,C 180,E1 23623.898,E2 23623.898} C_VEL
LIN {X 0,Y 534.102,Z 845.493,A -85,B 0,C 180,E1 23621.795,E2 23621.795} C_VEL
LIN {X 0,Y 538.962,Z 803.065,A -85,B 0,C 180,E1 23617.885,E2 23617.885} C_VEL
LIN {X 0,Y 543.245,Z 768.162,A -85,B 0,C 180,E1 23614.605,E2 23614.605} C_VEL
LIN {X 0,Y 547.318,Z 735.283,A -85,B 0,C 180,E1 23611.447,E2 23611.447} C_VEL
LIN {X 0,Y 548.919,Z 722.411,A -85,B 0,C 180,E1 23610.182,E2 23610.182} C_VEL
LIN {X 0,Y 541.285,Z 703.462,A -85,B 0,C 180,E1 23607.147,E2 23607.147} C_VEL
LIN {X 0,Y 533.831,Z 685.771,A -85,B 0,C 180,E1 23604.1,E2 23604.1} C_VEL
LIN {X 0,Y 526.036,Z 668.164,A -85,B 0,C 180,E1 23600.821,E2 23600.821} C_VEL
LIN {X 0,Y 519.651,Z 654.352,A -85,B 0,C 180,E1 23598.047,E2 23598.047} C_VEL
LIN {X 0,Y 513.956,Z 642.204,A -85,B 0,C 180,E1 23595.458,E2 23595.458} C_VEL
LIN {X 0,Y 509.494,Z 633.101,A -85,B 0,C 180,E1 23593.39,E2 23593.39} C_VEL
LIN {X 0,Y 507.454,Z 628.852,A -85,B 0,C 180,E1 23592.402,E2 23592.402} C_VEL
LIN {X 0,Y 505.909,Z 625.266,A -85,B 0,C 180,E1 23591.573,E2 23591.573} C_VEL
LIN {X 0,Y 505.862,Z 624.962,A -85,B 0,C 180,E1 23591.285,E2 23591.285} C_VEL
LIN {X 0,Y 505.871,Z 624.964,A -85,B 0,C 180,E1 23587.724,E2 23587.724} C_VEL
LIN {X 0,Y 505.853,Z 624.964,A -85,B 0,C 180,E1 23584.194,E2 23584.194} C_VEL
LIN {X 0,Y 505.865,Z 624.96,A -85,B 0,C 180,E1 23580.68,E2 23580.68} C_VEL
LIN {X 0,Y 505.862,Z 624.971,A -85,B 0,C 180,E1 23577.168,E2 23577.168} C_VEL
LIN {X 0,Y 505.862,Z 624.966,A -85,B 0,C 180,E1 23573.645,E2 23573.645} C_VEL
LIN {X 0,Y 505.864,Z 624.961,A -85,B 0,C 180,E1 23570.098,E2 23570.098} C_VEL
LIN {X 0,Y 505.867,Z 624.959,A -85,B 0,C 180,E1 23566.512,E2 23566.512} C_VEL
LIN {X 0,Y 505.864,Z 624.96,A -85,B 0,C 180,E1 23563.064,E2 23563.064} C_VEL
LIN {X 0,Y 505.864,Z 624.961,A -85,B 0,C 180,E1 23559.532,E2 23559.532} C_VEL
LIN {X 0,Y 505.857,Z 624.961,A -85,B 0,C 180,E1 23556.096,E2 23556.096} C_VEL
LIN {X 0,Y 505.866,Z 624.956,A -85,B 0,C 180,E1 23552.554,E2 23552.554} C_VEL
LIN {X 0,Y 505.866,Z 624.957,A -85,B 0,C 180,E1 23548.943,E2 23548.943} C_VEL
LIN {X 0,Y 505.868,Z 624.956,A -85,B 0,C 180,E1 23545.439,E2 23545.439} C_VEL
LIN {X 0,Y 505.866,Z 624.959,A -85,B 0,C 180,E1 23541.873,E2 23541.873} C_VEL
LIN {X 0,Y 505.857,Z 624.958,A -85,B 0,C 180,E1 23538.383,E2 23538.383} C_VEL
LIN {X 0,Y 505.867,Z 624.957,A -85,B 0,C 180,E1 23534.798,E2 23534.798} C_VEL
LIN {X 0,Y 505.871,Z 624.94,A -85,B 0,C 180,E1 23531.31,E2 23531.31} C_VEL
LIN {X 0,Y 505.883,Z 625.142,A -85,B 0,C 180,E1 23528.813,E2 23528.813} C_VEL
LIN {X 0,Y 514.947,Z 649.112,A -85,B 0,C 180,E1 23526.31,E2 23526.31} C_VEL
LIN {X 0,Y 521.757,Z 670.122,A -85,B 0,C 180,E1 23524.216,E2 23524.216} C_VEL
LIN {X 0,Y 523.293,Z 676.054,A -85,B 0,C 180,E1 23523.648,E2 23523.648} C_VEL
LIN {X 0,Y 521.501,Z 715.114,A -85,B 0,C 180,E1 23520.726,E2 23520.726} C_VEL
LIN {X 0,Y 519.154,Z 761.879,A -85,B 0,C 180,E1 23517.199,E2 23517.199} C_VEL
LIN {X 0,Y 517.018,Z 809.808,A -85,B 0,C 180,E1 23513.657,E2 23513.657} C_VEL
LIN {X 0,Y 515.718,Z 850.266,A -85,B 0,C 180,E1 23510.824,E2 23510.824} C_VEL
LIN {X 0,Y 516.426,Z 858.169,A -85,B 0,C 180,E1 23510.676,E2 23510.676} C_VEL
LIN {X 0,Y 514.108,Z 1019.546,A -85,B 0,C 180,E1 23508.385,E2 23508.385} C_VEL
LIN {X 0,Y 513.997,Z 1028.922,A -85,B 0,C 180,E1 23508.175,E2 23508.175} C_VEL
LIN {X 0,Y 512.921,Z 1036.479,A -85,B 0,C 180,E1 23508.009,E2 23508.009} C_VEL
LIN {X 0,Y 507.587,Z 1052.044,A -85,B 0,C 180,E1 23507.637,E2 23507.637} C_VEL
LIN {X 0,Y 505.519,Z 1060.211,A -85,B 0,C 180,E1 23507.319,E2 23507.319} C_VEL
LIN {X 0,Y 505.321,Z 1062.229,A -85,B 0,C 180,E1 23507.218,E2 23507.218} C_VEL
LIN {X 0,Y 504.394,Z 1077.973,A -85,B 0,C 180,E1 23506.288,E2 23506.288} C_VEL
LIN {X 0,Y 503.349,Z 1092.562,A -85,B 0,C 180,E1 23505.2,E2 23505.2} C_VEL
LIN {X 0,Y 502.221,Z 1106.17,A -85,B 0,C 180,E1 23503.938,E2 23503.938} C_VEL
LIN {X 0,Y 501.112,Z 1118.219,A -85,B 0,C 180,E1 23502.56,E2 23502.56} C_VEL
LIN {X 0,Y 499.976,Z 1129.969,A -85,B 0,C 180,E1 23500.904,E2 23500.904} C_VEL
LIN {X 0,Y 499.049,Z 1139.569,A -85,B 0,C 180,E1 23499.222,E2 23499.222} C_VEL
LIN {X 0,Y 498.271,Z 1147.839,A -85,B 0,C 180,E1 23497.377,E2 23497.377} C_VEL
LIN {X 0,Y 497.693,Z 1154.511,A -85,B 0,C 180,E1 23495.417,E2 23495.417} C_VEL
LIN {X 0,Y 497.318,Z 1159.286,A -85,B 0,C 180,E1 23493.456,E2 23493.456} C_VEL
LIN {X 0,Y 497.105,Z 1162.35,A -85,B 0,C 180,E1 23491.439,E2 23491.439} C_VEL
LIN {X 0,Y 497.025,Z 1163.651,A -85,B 0,C 180,E1 23489.422,E2 23489.422} C_VEL
LIN {X 0,Y 497.065,Z 1163.232,A -85,B 0,C 180,E1 23487.347,E2 23487.347} C_VEL
LIN {X 0,Y 497.246,Z 1161.006,A -85,B 0,C 180,E1 23485.269,E2 23485.269} C_VEL
LIN {X 0,Y 497.567,Z 1157.097,A -85,B 0,C 180,E1 23483.305,E2 23483.305} C_VEL
LIN {X 0,Y 498.079,Z 1151.373,A -85,B 0,C 180,E1 23481.339,E2 23481.339} C_VEL
LIN {X 0,Y 498.787,Z 1144.14,A -85,B 0,C 180,E1 23479.488,E2 23479.488} C_VEL
LIN {X 0,Y 499.673,Z 1135.413,A -85,B 0,C 180,E1 23477.752,E2 23477.752} C_VEL
LIN {X 0,Y 500.711,Z 1125.228,A -85,B 0,C 180,E1 23476.134,E2 23476.134} C_VEL
LIN {X 0,Y 501.868,Z 1113.605,A -85,B 0,C 180,E1 23474.633,E2 23474.633} C_VEL
LIN {X 0,Y 503.087,Z 1100.443,A -85,B 0,C 180,E1 23473.249,E2 23473.249} C_VEL
LIN {X 0,Y 504.254,Z 1086.097,A -85,B 0,C 180,E1 23472.039,E2 23472.039} C_VEL
LIN {X 0,Y 505.313,Z 1070.644,A -85,B 0,C 180,E1 23471.002,E2 23471.002} C_VEL
LIN {X 0,Y 506.145,Z 1055.207,A -85,B 0,C 180,E1 23470.195,E2 23470.195} C_VEL
LIN {X 0,Y 506.781,Z 1038.292,A -85,B 0,C 180,E1 23469.536,E2 23469.536} C_VEL
LIN {X 0,Y 507.093,Z 1020.669,A -85,B 0,C 180,E1 23469.081,E2 23469.081} C_VEL
LIN {X 0,Y 508.954,Z 894.857,A -85,B 0,C 180,E1 23467.258,E2 23467.258} C_VEL
LIN {X 0,Y 509.413,Z 855.531,A -85,B 0,C 180,E1 23466.688,E2 23466.688} C_VEL
LIN {X 0,Y 508.797,Z 850.745,A -85,B 0,C 180,E1 23466.576,E2 23466.576} C_VEL
LIN {X 0,Y 510.459,Z 806.484,A -85,B 0,C 180,E1 23463.41,E2 23463.41} C_VEL
LIN {X 0,Y 512.773,Z 759.959,A -85,B 0,C 180,E1 23459.923,E2 23459.923} C_VEL
LIN {X 0,Y 515.269,Z 713.045,A -85,B 0,C 180,E1 23456.355,E2 23456.355} C_VEL
LIN {X 0,Y 516.885,Z 679.099,A -85,B 0,C 180,E1 23453.772,E2 23453.772} C_VEL
LIN {X 0,Y 510.187,Z 657.991,A -85,B 0,C 180,E1 23451.623,E2 23451.623} C_VEL
LIN {X 0,Y 502.832,Z 638.404,A -85,B 0,C 180,E1 23449.518,E2 23449.518} C_VEL
LIN {X 0,Y 497.925,Z 625.958,A -85,B 0,C 180,E1 23448.117,E2 23448.117} C_VEL
LIN {X 0,Y 497.952,Z 626.133,A -85,B 0,C 180,E1 23446.205,E2 23446.205} C_VEL
LIN {X 0,Y 499.136,Z 629.305,A -85,B 0,C 180,E1 23445.641,E2 23445.641} C_VEL
LIN {X 0,Y 500.14,Z 631.172,A -85,B 0,C 180,E1 23445.272,E2 23445.272} C_VEL
LIN {X 0,Y 506.329,Z 644.254,A -85,B 0,C 180,E1 23442.89,E2 23442.89} C_VEL
LIN {X 0,Y 507.736,Z 646.835,A -85,B 0,C 180,E1 23442.479,E2 23442.479} C_VEL
LIN {X 0,Y 526.088,Z 672.92,A -85,B 0,C 180,E1 23440.029,E2 23440.029} C_VEL
LIN {X 0,Y 540.54,Z 694.468,A -85,B 0,C 180,E1 23438.233,E2 23438.233} C_VEL
LIN {X 0,Y 527.912,Z 947.916,A -85,B 0,C 180,E1 23433.822,E2 23433.822} C_VEL
LIN {X 0,Y 526.623,Z 976.828,A -85,B 0,C 180,E1 23433.238,E2 23433.238} C_VEL
LIN {X 0,Y 525.192,Z 999.191,A -85,B 0,C 180,E1 23432.602,E2 23432.602} C_VEL
LIN {X 0,Y 523.318,Z 1020.975,A -85,B 0,C 180,E1 23431.783,E2 23431.783} C_VEL
LIN {X 0,Y 520.929,Z 1044.01,A -85,B 0,C 180,E1 23430.702,E2 23430.702} C_VEL
LIN {X 0,Y 518.488,Z 1064.704,A -85,B 0,C 180,E1 23429.52,E2 23429.52} C_VEL
LIN {X 0,Y 515.828,Z 1084.474,A -85,B 0,C 180,E1 23428.165,E2 23428.165} C_VEL
LIN {X 0,Y 512.941,Z 1104.18,A -85,B 0,C 180,E1 23426.575,E2 23426.575} C_VEL
LIN {X 0,Y 510.257,Z 1121.84,A -85,B 0,C 180,E1 23424.917,E2 23424.917} C_VEL
LIN {X 0,Y 507.582,Z 1138.478,A -85,B 0,C 180,E1 23423.08,E2 23423.08} C_VEL
LIN {X 0,Y 504.971,Z 1154.732,A -85,B 0,C 180,E1 23421.002,E2 23421.002} C_VEL
LIN {X 0,Y 502.775,Z 1168.776,A -85,B 0,C 180,E1 23418.915,E2 23418.915} C_VEL
LIN {X 0,Y 500.859,Z 1181.425,A -85,B 0,C 180,E1 23416.707,E2 23416.707} C_VEL
LIN {X 0,Y 499.28,Z 1192.888,A -85,B 0,C 180,E1 23414.379,E2 23414.379} C_VEL
LIN {X 0,Y 498.029,Z 1202.904,A -85,B 0,C 180,E1 23411.935,E2 23411.935} C_VEL
LIN {X 0,Y 497.141,Z 1211.543,A -85,B 0,C 180,E1 23409.376,E2 23409.376} C_VEL
LIN {X 0,Y 496.604,Z 1218.187,A -85,B 0,C 180,E1 23406.939,E2 23406.939} C_VEL
LIN {X 0,Y 496.274,Z 1223.446,A -85,B 0,C 180,E1 23404.391,E2 23404.391} C_VEL
LIN {X 0,Y 496.129,Z 1227.264,A -85,B 0,C 180,E1 23401.848,E2 23401.848} C_VEL
LIN {X 0,Y 496.073,Z 1229.424,A -85,B 0,C 180,E1 23399.307,E2 23399.307} C_VEL
LIN {X 0,Y 496.072,Z 1230.237,A -85,B 0,C 180,E1 23396.765,E2 23396.765} C_VEL
LIN {X 0,Y 496.103,Z 1229.461,A -85,B 0,C 180,E1 23394.216,E2 23394.216} C_VEL
LIN {X 0,Y 496.182,Z 1227.095,A -85,B 0,C 180,E1 23391.541,E2 23391.541} C_VEL
LIN {X 0,Y 496.38,Z 1223.499,A -85,B 0,C 180,E1 23389.085,E2 23389.085} C_VEL
LIN {X 0,Y 496.78,Z 1218.065,A -85,B 0,C 180,E1 23386.498,E2 23386.498} C_VEL
LIN {X 0,Y 497.439,Z 1211.364,A -85,B 0,C 180,E1 23384.015,E2 23384.015} C_VEL
LIN {X 0,Y 498.406,Z 1203.178,A -85,B 0,C 180,E1 23381.61,E2 23381.61} C_VEL
LIN {X 0,Y 499.805,Z 1192.883,A -85,B 0,C 180,E1 23379.111,E2 23379.111} C_VEL
LIN {X 0,Y 501.561,Z 1181.276,A -85,B 0,C 180,E1 23376.751,E2 23376.751} C_VEL
LIN {X 0,Y 503.548,Z 1168.659,A -85,B 0,C 180,E1 23374.601,E2 23374.601} C_VEL
LIN {X 0,Y 505.935,Z 1153.878,A -85,B 0,C 180,E1 23372.454,E2 23372.454} C_VEL
LIN {X 0,Y 508.317,Z 1139.219,A -85,B 0,C 180,E1 23370.624,E2 23370.624} C_VEL
LIN {X 0,Y 510.719,Z 1123.373,A -85,B 0,C 180,E1 23368.943,E2 23368.943} C_VEL
LIN {X 0,Y 513.284,Z 1105.318,A -85,B 0,C 180,E1 23367.305,E2 23367.305} C_VEL
LIN {X 0,Y 515.538,Z 1088.108,A -85,B 0,C 180,E1 23365.975,E2 23365.975} C_VEL
LIN {X 0,Y 517.598,Z 1069.475,A -85,B 0,C 180,E1 23364.777,E2 23364.777} C_VEL
LIN {X 0,Y 519.422,Z 1049.391,A -85,B 0,C 180,E1 23363.705,E2 23363.705} C_VEL
LIN {X 0,Y 520.852,Z 1029.648,A -85,B 0,C 180,E1 23362.854,E2 23362.854} C_VEL
LIN {X 0,Y 521.802,Z 1008.598,A -85,B 0,C 180,E1 23362.159,E2 23362.159} C_VEL
LIN {X 0,Y 522.299,Z 987.357,A -85,B 0,C 180,E1 23361.658,E2 23361.658} C_VEL
LIN {X 0,Y 523.562,Z 936.928,A -85,B 0,C 180,E1 23360.823,E2 23360.823} C_VEL
LIN {X 0,Y 526.703,Z 870.489,A -85,B 0,C 180,E1 23359.644,E2 23359.644} C_VEL
LIN {X 0,Y 531.211,Z 807.07,A -85,B 0,C 180,E1 23358.372,E2 23358.372} C_VEL
LIN {X 0,Y 533.35,Z 782.802,A -85,B 0,C 180,E1 23357.849,E2 23357.849} C_VEL
LIN {X 0,Y 529.161,Z 786.838,A -85,B 0,C 180,E1 23357.232,E2 23357.232} C_VEL
LIN {X 0,Y 522.101,Z 798.683,A -85,B 0,C 180,E1 23356.043,E2 23356.043} C_VEL
LIN {X 0,Y 517.527,Z 809.841,A -85,B 0,C 180,E1 23354.866,E2 23354.866} C_VEL
LIN {X 0,Y 514.909,Z 821.897,A -85,B 0,C 180,E1 23353.658,E2 23353.658} C_VEL
LIN {X 0,Y 514.174,Z 835.549,A -85,B 0,C 180,E1 23352.399,E2 23352.399} C_VEL
LIN {X 0,Y 515.57,Z 850.714,A -85,B 0,C 180,E1 23351.075,E2 23351.075} C_VEL
LIN {X 0,Y 519.337,Z 866.869,A -85,B 0,C 180,E1 23349.713,E2 23349.713} C_VEL
LIN {X 0,Y 525.929,Z 886.003,A -85,B 0,C 180,E1 23348.239,E2 23348.239} C_VEL
LIN {X 0,Y 534.107,Z 902.742,A -85,B 0,C 180,E1 23346.973,E2 23346.973} C_VEL
LIN {X 0,Y 537.82,Z 909.365,A -85,B 0,C 180,E1 23346.492,E2 23346.492} C_VEL
LIN {X 0,Y 531.922,Z 927.93,A -85,B 0,C 180,E1 23346.552,E2 23346.552} C_VEL
LIN {X 0,Y 526.415,Z 947.573,A -85,B 0,C 180,E1 23346.457,E2 23346.457} C_VEL
LIN {X 0,Y 522.803,Z 964.751,A -85,B 0,C 180,E1 23346.198,E2 23346.198} C_VEL
LIN {X 0,Y 520.603,Z 981.228,A -85,B 0,C 180,E1 23345.792,E2 23345.792} C_VEL
LIN {X 0,Y 517.19,Z 1016.966,A -85,B 0,C 180,E1 23344.64,E2 23344.64} C_VEL
LIN {X 0,Y 514.126,Z 1048.686,A -85,B 0,C 180,E1 23343.395,E2 23343.395} C_VEL
LIN {X 0,Y 511.366,Z 1079.214,A -85,B 0,C 180,E1 23341.961,E2 23341.961} C_VEL
LIN {X 0,Y 508.944,Z 1107.444,A -85,B 0,C 180,E1 23340.404,E2 23340.404} C_VEL
LIN {X 0,Y 506.74,Z 1133.718,A -85,B 0,C 180,E1 23338.717,E2 23338.717} C_VEL
LIN {X 0,Y 504.751,Z 1157.905,A -85,B 0,C 180,E1 23336.921,E2 23336.921} C_VEL
LIN {X 0,Y 502.971,Z 1179.548,A -85,B 0,C 180,E1 23335.053,E2 23335.053} C_VEL
LIN {X 0,Y 501.378,Z 1198.824,A -85,B 0,C 180,E1 23333.135,E2 23333.135} C_VEL
LIN {X 0,Y 500.068,Z 1215.347,A -85,B 0,C 180,E1 23331.219,E2 23331.219} C_VEL
LIN {X 0,Y 498.899,Z 1230.41,A -85,B 0,C 180,E1 23329.19,E2 23329.19} C_VEL
LIN {X 0,Y 497.926,Z 1243.972,A -85,B 0,C 180,E1 23327.05,E2 23327.05} C_VEL
LIN {X 0,Y 497.214,Z 1255.326,A -85,B 0,C 180,E1 23324.918,E2 23324.918} C_VEL
LIN {X 0,Y 496.667,Z 1265.209,A -85,B 0,C 180,E1 23322.677,E2 23322.677} C_VEL
LIN {X 0,Y 496.327,Z 1273.606,A -85,B 0,C 180,E1 23320.33,E2 23320.33} C_VEL
LIN {X 0,Y 496.135,Z 1280.107,A -85,B 0,C 180,E1 23317.995,E2 23317.995} C_VEL
LIN {X 0,Y 496.068,Z 1285.046,A -85,B 0,C 180,E1 23315.554,E2 23315.554} C_VEL
LIN {X 0,Y 496.057,Z 1288.251,A -85,B 0,C 180,E1 23313.121,E2 23313.121} C_VEL
LIN {X 0,Y 496.049,Z 1289.701,A -85,B 0,C 180,E1 23310.695,E2 23310.695} C_VEL
LIN {X 0,Y 496.038,Z 1289.544,A -85,B 0,C 180,E1 23308.269,E2 23308.269} C_VEL
LIN {X 0,Y 496.019,Z 1287.774,A -85,B 0,C 180,E1 23305.84,E2 23305.84} C_VEL
LIN {X 0,Y 496.03,Z 1284.168,A -85,B 0,C 180,E1 23303.288,E2 23303.288} C_VEL
LIN {X 0,Y 496.139,Z 1279.094,A -85,B 0,C 180,E1 23300.841,E2 23300.841} C_VEL
LIN {X 0,Y 496.445,Z 1271.902,A -85,B 0,C 180,E1 23298.265,E2 23298.265} C_VEL
LIN {X 0,Y 496.974,Z 1263.251,A -85,B 0,C 180,E1 23295.793,E2 23295.793} C_VEL
LIN {X 0,Y 497.872,Z 1252.081,A -85,B 0,C 180,E1 23293.192,E2 23293.192} C_VEL
LIN {X 0,Y 499.089,Z 1239.93,A -85,B 0,C 180,E1 23290.82,E2 23290.82} C_VEL
LIN {X 0,Y 500.721,Z 1225.679,A -85,B 0,C 180,E1 23288.445,E2 23288.445} C_VEL
LIN {X 0,Y 502.84,Z 1208.986,A -85,B 0,C 180,E1 23286.07,E2 23286.07} C_VEL
LIN {X 0,Y 505.289,Z 1191.093,A -85,B 0,C 180,E1 23283.88,E2 23283.88} C_VEL
LIN {X 0,Y 508.123,Z 1171.622,A -85,B 0,C 180,E1 23281.82,E2 23281.82} C_VEL
LIN {X 0,Y 511.061,Z 1151.718,A -85,B 0,C 180,E1 23280.01,E2 23280.01} C_VEL
LIN {X 0,Y 514.268,Z 1130.674,A -85,B 0,C 180,E1 23278.337,E2 23278.337} C_VEL
LIN {X 0,Y 517.525,Z 1108.737,A -85,B 0,C 180,E1 23276.856,E2 23276.856} C_VEL
LIN {X 0,Y 520.967,Z 1085.69,A -85,B 0,C 180,E1 23275.517,E2 23275.517} C_VEL
LIN {X 0,Y 524.175,Z 1062.902,A -85,B 0,C 180,E1 23274.425,E2 23274.425} C_VEL
LIN {X 0,Y 527.405,Z 1038.995,A -85,B 0,C 180,E1 23273.468,E2 23273.468} C_VEL
LIN {X 0,Y 530.37,Z 1014.569,A -85,B 0,C 180,E1 23272.712,E2 23272.712} C_VEL
LIN {X 0,Y 532.8,Z 988.936,A -85,B 0,C 180,E1 23272.087,E2 23272.087} C_VEL
LIN {X 0,Y 534.577,Z 968.902,A -85,B 0,C 180,E1 23271.738,E2 23271.738} C_VEL
LIN {X 0,Y 538.499,Z 944.6,A -85,B 0,C 180,E1 23271.5,E2 23271.5} C_VEL
LIN {X 0,Y 539.097,Z 943.048,A -85,B 0,C 180,E1 23271.453,E2 23271.453} C_VEL
LIN {X 0,Y 544.773,Z 933.561,A -85,B 0,C 180,E1 23270.931,E2 23270.931} C_VEL
LIN {X 0,Y 537.054,Z 918.955,A -85,B 0,C 180,E1 23269.104,E2 23269.104} C_VEL
LIN {X 0,Y 531.35,Z 903.005,A -85,B 0,C 180,E1 23267.212,E2 23267.212} C_VEL
LIN {X 0,Y 527.864,Z 886.351,A -85,B 0,C 180,E1 23265.354,E2 23265.354} C_VEL
LIN {X 0,Y 526.436,Z 868.035,A -85,B 0,C 180,E1 23263.438,E2 23263.438} C_VEL
LIN {X 0,Y 527.231,Z 846.401,A -85,B 0,C 180,E1 23261.325,E2 23261.325} C_VEL
LIN {X 0,Y 532.153,Z 805.258,A -85,B 0,C 180,E1 23257.502,E2 23257.502} C_VEL
LIN {X 0,Y 536.507,Z 770.955,A -85,B 0,C 180,E1 23254.253,E2 23254.253} C_VEL
LIN {X 0,Y 540.781,Z 738.007,A -85,B 0,C 180,E1 23251.055,E2 23251.055} C_VEL
LIN {X 0,Y 542.192,Z 726.029,A -85,B 0,C 180,E1 23249.863,E2 23249.863} C_VEL
LIN {X 0,Y 534.592,Z 707.115,A -85,B 0,C 180,E1 23246.793,E2 23246.793} C_VEL
LIN {X 0,Y 527.416,Z 690.062,A -85,B 0,C 180,E1 23243.817,E2 23243.817} C_VEL
LIN {X 0,Y 519.931,Z 672.973,A -85,B 0,C 180,E1 23240.606,E2 23240.606} C_VEL
LIN {X 0,Y 513.292,Z 658.662,A -85,B 0,C 180,E1 23237.691,E2 23237.691} C_VEL
LIN {X 0,Y 508.091,Z 647.478,A -85,B 0,C 180,E1 23235.29,E2 23235.29} C_VEL
